// TIA Portal project "KWT_80621" (V14)

(* hardware
DEVICE "S7-1200-Station_1"  S7-1200 Station
   slot 0: "Baugruppenträger_0"  S7-1200 Rack  Rack  V1.0
   slot 1: "PLC_1"  CPU 1214C DC/DC/DC  6ES7 214-1AG40-0XB0  V4.2
   slot 2: "DI 16/DQ 16x24VDC_1"  6ES7 223-1BL32-0XB0  V2.0
   slot 3: "DI 16x24VDC_1"  6ES7 221-1BH32-0XB0  V2.0
   slot 4: "AI 4x13BIT_1"  6ES7 231-4HD32-0XB0  V2.0
   slot 5: "AQ 4x14BIT_1"  6ES7 232-4HD32-0XB0  V2.0
DEVICE "HMI_1"  KTP1200 Basic PN
   slot 0: "KTP1200 Basic PN"  KTP1200 Basic PN  6AV2 123-2MB03-0AX0  14.0.1.0
   slot 1: "HMI_RT_1"  KTP1200 Basic PN  6AV2 123-2MB03-0AX0  14.0.1.0
   slot 5: "HMI_1.IE_CP_1"  PROFINET Interface  14.0.1.0
      slot 1: "PROFINET Schnittstelle_1"  PROFINET Interface
         slot 1: "Port_1"  Port
*)

// ===== PLC "PLC_1"  CPU 1214C DC/DC/DC =====

VAR_GLOBAL   // PLC tag table "Default tag table"
   "System_Byte" AT %MB1 : Byte;
   "FirstScan" AT %M1.0 : Bool;
   "DiagStatusUpdate" AT %M1.1 : Bool;
   "AlwaysTRUE" AT %M1.2 : Bool;
   "AlwaysFALSE" AT %M1.3 : Bool;
   "Clock_Byte" AT %MB0 : Byte;
   "Clock_10Hz" AT %M0.0 : Bool;
   "Clock_5Hz" AT %M0.1 : Bool;
   "Clock_2.5Hz" AT %M0.2 : Bool;
   "Clock_2Hz" AT %M0.3 : Bool;
   "Clock_1.25Hz" AT %M0.4 : Bool;
   "Clock_1Hz" AT %M0.5 : Bool;
   "Clock_0.625Hz" AT %M0.6 : Bool;
   "Clock_0.5Hz" AT %M0.7 : Bool;
END_VAR

VAR_GLOBAL CONSTANT   // PLC tag table "Default tag table"
   "MaxAI10Bit" : Int := 27648;   // AI Max 10 Bit
END_VAR

VAR_GLOBAL   // PLC tag table "1~DI_14_DQ_10"
   "Steuerspannung Ein" AT %I0.0 : Bool;
   "Sicherung Ausgänge OK" AT %I0.1 : Bool;
   "KT 1 Ventilator Störung" AT %I0.2 : Bool;   // Kühlturm 1 Ventilator Störung
   "KT 1 Ventilator Betrieb" AT %I0.3 : Bool;   // Kühlturm 1 Ventilator Betrieb
   "KT 1 Ventilator RS" AT %I0.4 : Bool;   // Kühlturm 1 Ventilator Reparaturschalter ein
   "KT 2 Ventilator Störung" AT %I0.5 : Bool;   // Kühlturm 2 Ventilator Störung
   "KT 2 Ventilator Betrieb" AT %I0.6 : Bool;   // Kühlturm 2 Ventilator Betrieb
   "KT 2 Ventilator RS" AT %I0.7 : Bool;   // Kühlturm 2 Ventilator Reparaturschalter ein
   "Werkspumpe 1 Störung" AT %I1.0 : Bool;
   "Werkspumpe 1 Betrieb" AT %I1.1 : Bool;
   "Werkspumpe 2 Störung" AT %I1.2 : Bool;
   "Werkspumpe 2 Betrieb" AT %I1.3 : Bool;
   "Reserve DI1.4" AT %I1.4 : Bool;
   "Reserve DI1.5" AT %I1.5 : Bool;
   "KT 1 Ventilator" AT %Q0.0 : Bool;   // Kühlturm 1 Ventilator
   "KT 2 Ventilator" AT %Q0.1 : Bool;   // Kühlturm 2 Ventilator
   "Werkspumpe 1" AT %Q0.2 : Bool;
   "Werkspumpe 2" AT %Q0.3 : Bool;
   "Kühlwasserpumpe 1" AT %Q0.4 : Bool;
   "Kühlwasserpumpe 2" AT %Q0.5 : Bool;
   "Rundumleuchte Störung" AT %Q0.6 : Bool;
   "Reserve DQ0.7" AT %Q0.7 : Bool;
   "KT 1 Sprührohr-Klappen öffnen" AT %Q1.0 : Bool;   // Kühlturm 1
   "KT 2 Sprührohr-Klappen öffnen" AT %Q1.1 : Bool;   // Kühlturm 2
END_VAR

VAR_GLOBAL   // PLC tag table "2~DI_16_DQ_16x24VDC"
   "Kühlwasserpumpe 1 MSS OK" AT %I8.0 : Bool;   // Kühlwasserpumpe 1 Motorschutzschalter
   "Kühlwasserpumpe 2 MSS OK" AT %I8.1 : Bool;   // Kühlwasserpumpe 2 Motorschutzschalter
   "Ofenpumpe 1 MSS OK" AT %I8.2 : Bool;   // Ofenpumpe 1 Motorschutzschalter
   "Ofenpumpe 2 MSS OK" AT %I8.3 : Bool;   // Ofenpumpe 2 Motorschutzschalter
   "Kühlwasserpumpe 1 Betrieb" AT %I8.4 : Bool;
   "Kühlwasserpumpe 2 Betrieb" AT %I8.5 : Bool;
   "Ofenpumpe 1 Betrieb" AT %I8.6 : Bool;
   "Ofenpumpe 2 Betrieb" AT %I8.7 : Bool;
   "KT 1 Sprührohr-Klappen geöffnet" AT %I9.0 : Bool;   // Kühlturm 1
   "KT 2 Sprührohr-Klappen geöffnet" AT %I9.1 : Bool;   // Kühlturm 2
   "HA 1 Klappe geöffnet" AT %I9.2 : Bool;   // Hebeanlage 1 Klappe geöffnet
   "HA 1 Klappe geschlossen" AT %I9.3 : Bool;   // Hebeanlage 1 Klappe geschlossen Option
   "HA 2 Klappe geöffnet" AT %I9.4 : Bool;   // Hebeanlage 2 Klappe geöffnet
   "HA 2 Klappe geschlossen" AT %I9.5 : Bool;   // Hebeanlage 2 Klappe geschlossen Option
   "Reserve DI9.6" AT %I9.6 : Bool;
   "Reserve DI9.7" AT %I9.7 : Bool;
   "HA 1 Klappe Freigabe" AT %Q8.0 : Bool;   // Hebeanlage 1 Klappe Freigabe
   "HA 2 Klappe Freigabe" AT %Q8.1 : Bool;   // Hebeanlage 2 Klappe Freigabe
   "Ofenpumpe 1" AT %Q8.2 : Bool;
   "Ofenpumpe 2" AT %Q8.3 : Bool;
   "Reserve DQ8.4" AT %Q8.4 : Bool;
   "Reserve DQ8.5" AT %Q8.5 : Bool;
   "Reserve DQ8.6" AT %Q8.6 : Bool;
   "Reserve DQ8.7" AT %Q8.7 : Bool;
   "WSB Magnetventil" AT %Q9.0 : Bool;   // Wasserstation Behälter Magnetventil Nachfüllung
   "Reserve DQ9.1" AT %Q9.1 : Bool;
   "Reserve DQ9.2" AT %Q9.2 : Bool;
   "Reserve DQ9.3" AT %Q9.3 : Bool;
   "Reserve DQ9.4" AT %Q9.4 : Bool;
   "Reserve DQ9.5" AT %Q9.5 : Bool;
   "Reserve DQ9.6" AT %Q9.6 : Bool;
   "Reserve DQ9.7" AT %Q9.7 : Bool;
END_VAR

VAR_GLOBAL   // PLC tag table "3~DI_16x24VDC"
   "Absalzanlage läuft" AT %I12.0 : Bool;   // Absalzanlage Umwälzpumpe läuft
   "WSB OUT1" AT %I12.1 : Bool;   // Wasserstation Behälter Füllstand binär Bit 0
   "WSB OUT2" AT %I12.2 : Bool;   // Wasserstation Behälter Füllstand binär Bit 1
   "WSB OUT3" AT %I12.3 : Bool;   // Wasserstation Behälter Füllstand binär Bit 2
   "WSB OUT4" AT %I12.4 : Bool;   // Wasserstation Behälter Füllstand binär Bit 3
   "Reserve DI12.5" AT %I12.5 : Bool;
   "Reserve DI12.6" AT %I12.6 : Bool;
   "Reserve DI12.7" AT %I12.7 : Bool;
   "Reserve DI13.0" AT %I13.0 : Bool;
   "Reserve DI13.1" AT %I13.1 : Bool;
   "Reserve DI13.2" AT %I13.2 : Bool;
   "Reserve DI13.3" AT %I13.3 : Bool;
   "Reserve DI13.4" AT %I13.4 : Bool;
   "Reserve DI13.5" AT %I13.5 : Bool;
   "Reserve DI13.6" AT %I13.6 : Bool;
   "Reserve DI13.7" AT %I13.7 : Bool;
   "WSB OUT1 M" AT %M12.0 : Bool;   // Wasserstation Behälter Füllstand binär Bit 0
   "WSB OUT2 M" AT %M12.1 : Bool;   // Wasserstation Behälter Füllstand binär Bit 1
   "WSB OUT3 M" AT %M12.2 : Bool;   // Wasserstation Behälter Füllstand binär Bit 2
   "WSB OUT4 M" AT %M12.3 : Bool;   // Wasserstation Behälter Füllstand binär Bit 3
   "WSB OUT Byte" AT %MB12 : Byte;   // Wasserstation Behälter Füllstand binär Byte
END_VAR

VAR_GLOBAL   // PLC tag table "4~AI_4x13BIT"
   "HA 1 Differenzdruck" AT %IW128 : Int;   // Hebeanlage 1 Differenzdruck Filter
   "HA 2 Differenzdruck" AT %IW130 : Int;   // Hebeanlage 2 Differenzdruck Filter
   "Reserve IW132" AT %IW132 : Int;
   "Reserve IW134" AT %IW134 : Int;
END_VAR

VAR_GLOBAL   // PLC tag table "5~AQ_4"
   "KT 1 Ventilator Sollwert" AT %QW144 : Int;   // Kühlturm 1 Sollwert
   "KT 2 Ventilator Sollwert" AT %QW146 : Int;   // Kühlturm 2 Sollwert
   "HA 1 Klappe Durchflußmenge" AT %QW148 : Int;   // Hebeanlage 1 Klappe Durchflußmenge
   "HA 2 Klappe Durchflußmenge" AT %QW150 : Int;   // Hebeanlage 2 Klappe Durchflußmenge
END_VAR

VAR_GLOBAL   // PLC tag table "1~AI_2"
   "Vorlauftemperatur Werk" AT %IW64 : Int;
   "Vorlauftemperatur Ofen" AT %IW66 : Int;
END_VAR

TYPE "RTM_MODE"
   STRUCT
      FETCH : Byte := 16#0;   // 0: Read out (the status is then written to CQ and the current value to CV). After the operating hours counter has reached (2^31) - 1 hours, it stops at the highest value that can be displayed and outputs an "Overflow" error message.
      START : Byte := 16#1;   // 1: start (at the last counter value)
      STOP : Byte := 16#2;   // 2: stop
      SET : Byte := 16#4;   // 4: set to the value specified in the parameter PV
      SET_START : Byte := 16#5;   // 5: set to the value specified in the parameter PV and start
      SET_STOP : Byte := 16#6;   // 6: set to the value specified in the parameter PV and stop
      SAVE_MC : Byte := 16#7;   // 7: save all RTM values in the CPU to the MC (Memory Card)
   END_STRUCT;
END_TYPE

DATA_BLOCK "Main_DB"   // DB1
{ S7_Optimized_Access := 'TRUE' }
AUTHOR : Searinox(Gerrit_Vogtlaender)
FAMILY : AKK
VERSION : 0.1
// stored: InstanceOfName MainInstane
"MainInstane"
BEGIN
END_DATA_BLOCK

DATA_BLOCK "Retain_DB"   // DB2
{ S7_Optimized_Access := 'TRUE' }
AUTHOR : Searinox
VERSION : 0.1
   VAR RETAIN
      Settings : Struct
         MaxPressureDeltaPerc1 : Int := 50;   // Maximum pressure difference in percent before alarm
         MaxPressureDeltaPerc2 : Int := 50;   // Maximum pressure difference in percent before alarm
         MaxTempTransgression : Real := 4.0;   // Maximum temperature overrun of setpoint in centigrade before alarm
      END_STRUCT;
   END_VAR
BEGIN
END_DATA_BLOCK

FUNCTION_BLOCK "MainInstane"   // FB1, SCL
{ S7_Optimized_Access := 'TRUE' }
AUTHOR : Searinox(Gerrit_Vogtlaender)
FAMILY : AKK
VERSION : 0.1
   VAR
      AlwaysRUN : "AlwaysRUN";
      Auto : "Auto";
      Hand : "Hand";
      AutoMode : Bool := true;
      FlowTemperaturePlant : Real;
      FlowTemperatureFurnace : Real;
   END_VAR
   VAR RETAIN
      HMI : Struct
         StorageTankLevel : Struct
            P1 : Int := 14;   // position 1, e.g. maximum value reached
            P2 : Int := 6;   // position 2, e.g. upper preset value reached
            P3 : Int := 4;   // position 3, e.g. lower preset value reached
            P4 : Int := 2;   // position 4, e.g. minimum value reached
         END_STRUCT;
         StorageTankRefill : Bool;
      END_STRUCT;
   END_VAR
BEGIN
   #AlwaysRUN();

   IF NOT "Steuerspannung Ein" OR NOT "Sicherung Ausgänge OK" THEN
       #AutoMode := 0;
       "KT 1 Ventilator" := 0;
       "KT 2 Ventilator" := 0;
       "Werkspumpe 1" := 0;
       "Werkspumpe 2" := 0;
       "Kühlwasserpumpe 1" := 0;
       "Kühlwasserpumpe 2" := 0;
       //"Rundumleuchte Störung" := 0;
       "Reserve DQ0.7" := 0;
       "KT 1 Sprührohr-Klappen öffnen" := 0;
       "KT 2 Sprührohr-Klappen öffnen" := 0;
       "HA 1 Klappe Freigabe" := 0;
       "HA 2 Klappe Freigabe" := 0;
       "Ofenpumpe 1" := 0;
       "Ofenpumpe 2" := 0;
       "Reserve DQ8.4" := 0;
       "Reserve DQ8.5" := 0;
       "Reserve DQ8.6" := 0;
       "Reserve DQ8.7" := 0;
       "WSB Magnetventil" := 0;
       "Reserve DQ9.1" := 0;
       "Reserve DQ9.2" := 0;
       "Reserve DQ9.3" := 0;
       "Reserve DQ9.4" := 0;
       "Reserve DQ9.5" := 0;
       "Reserve DQ9.6" := 0;
       "Reserve DQ9.7" := 0;
   END_IF;

   IF #AutoMode THEN
       #Auto();
   ELSE
       #Hand();
   END_IF;
END_FUNCTION_BLOCK

FUNCTION_BLOCK "Alarm"   // FB2, SCL
{ S7_Optimized_Access := 'TRUE' }
AUTHOR : Searinox
VERSION : 0.1
   VAR
      "Steuerspannung Ein" : Int;
      "Sicherung Ausgänge OK" : Int;
      "KT 1 Ventilator Störung" : Int;
      "KT 1 Ventilator RS" : Int;
      "KT 2 Ventilator Störung" : Int;
      "KT 2 Ventilator RS" : Int;
      "Werkspumpe 1 Störung" : Int;
      "Werkspumpe 2 Störung" : Int;
      "Kühlwasserpumpe 1 MSS OK" : Int;
      "Kühlwasserpumpe 2 MSS OK" : Int;
      "Ofenpumpe 1 MSS OK" : Int;
      "Ofenpumpe 2 MSS OK" : Int;
      s_alarms : Int;
      FlowTemperaturePlant : Int;
      FlowTemperatureFurnace : Int;
      "HA 1 Differenzdruck" : Int;
      "HA 2 Differenzdruck" : Int;
      SurgeTankRunDry : Int;
      SurgeTankOverflow : Int;
   END_VAR
   VAR_TEMP
      PressureDeltaPerc1 : Int;
      PressureDeltaPerc2 : Int;
   END_VAR
BEGIN
   REGION bool
       #"Steuerspannung Ein" := BOOL_TO_INT(NOT "Steuerspannung Ein");
       #"Sicherung Ausgänge OK" := BOOL_TO_INT(NOT "Sicherung Ausgänge OK");
       #"KT 1 Ventilator Störung" := BOOL_TO_INT("KT 1 Ventilator Störung");
       #"KT 2 Ventilator Störung" := BOOL_TO_INT("KT 2 Ventilator Störung");
       #"KT 1 Ventilator RS" := BOOL_TO_INT(NOT "KT 1 Ventilator RS");
       #"KT 2 Ventilator RS" := BOOL_TO_INT(NOT "KT 2 Ventilator RS");
       #"Werkspumpe 1 Störung" := BOOL_TO_INT("Werkspumpe 1 Störung");
       #"Werkspumpe 2 Störung" := BOOL_TO_INT("Werkspumpe 2 Störung");
       #"Kühlwasserpumpe 1 MSS OK" := BOOL_TO_INT(NOT "Kühlwasserpumpe 1 MSS OK");
       #"Kühlwasserpumpe 2 MSS OK" := BOOL_TO_INT(NOT "Kühlwasserpumpe 2 MSS OK");
       #"Ofenpumpe 1 MSS OK" := BOOL_TO_INT(NOT "Ofenpumpe 1 MSS OK");
       #"Ofenpumpe 2 MSS OK" := BOOL_TO_INT(NOT "Ofenpumpe 2 MSS OK");
   END_REGION
   REGION analog
       // temperatures
       #FlowTemperaturePlant := BOOL_TO_INT("Main_DB".FlowTemperaturePlant >= ("Main_DB".Auto.s_Max + "Retain_DB".Settings.MaxTempTransgression));
       #FlowTemperatureFurnace := BOOL_TO_INT("Main_DB".FlowTemperatureFurnace >= ("Main_DB".Auto.s_Max + "Retain_DB".Settings.MaxTempTransgression));
       // pressures
       #PressureDeltaPerc1 := "ScaleValueInt"(VALUE := "HA 1 Differenzdruck",
                                                XMIN := 0, XMAX := "MaxAI10Bit",
                                                YMIN := 0, YMAX := 100);
       #"HA 1 Differenzdruck" := BOOL_TO_INT(#PressureDeltaPerc1 >= "Retain_DB".Settings.MaxPressureDeltaPerc1);
       #PressureDeltaPerc2 := "ScaleValueInt"(VALUE := "HA 2 Differenzdruck",
                                                XMIN := 0, XMAX := "MaxAI10Bit",
                                                YMIN := 0, YMAX := 100);
       #"HA 2 Differenzdruck" := BOOL_TO_INT(#PressureDeltaPerc2 >= "Retain_DB".Settings.MaxPressureDeltaPerc2);

       #SurgeTankRunDry := BOOL_TO_INT("WSB OUT Byte" <= "Main_DB".HMI.StorageTankLevel.P4);
       #SurgeTankOverflow := BOOL_TO_INT("WSB OUT Byte" >= "Main_DB".HMI.StorageTankLevel.P1);
   END_REGION

   #s_alarms := 0;
   #s_alarms += #"Steuerspannung Ein";
   #s_alarms += #"Sicherung Ausgänge OK";
   #s_alarms += #"KT 1 Ventilator Störung";
   #s_alarms += #"KT 1 Ventilator RS";
   #s_alarms += #"KT 2 Ventilator Störung";
   #s_alarms += #"KT 2 Ventilator RS";
   #s_alarms += #"Werkspumpe 1 Störung";
   #s_alarms += #"Werkspumpe 2 Störung";
   #s_alarms += #"Kühlwasserpumpe 1 MSS OK";
   #s_alarms += #"Kühlwasserpumpe 2 MSS OK";
   #s_alarms += #"Ofenpumpe 1 MSS OK";
   #s_alarms += #"Ofenpumpe 2 MSS OK";
   #s_alarms += #FlowTemperaturePlant;
   #s_alarms += #FlowTemperatureFurnace;
   #s_alarms += #"HA 1 Differenzdruck";
   #s_alarms += #"HA 2 Differenzdruck";
   #s_alarms += #SurgeTankRunDry;
   #s_alarms += #SurgeTankOverflow;

   "Rundumleuchte Störung" := #s_alarms > 0;


   // heizung klappen & endschalter offen zu 
   //Trockenlauf & Überlauf
   //ZU-Klappen 1 geöffnet
END_FUNCTION_BLOCK

FUNCTION_BLOCK "AlwaysRUN"   // FB10, SCL
{ S7_Optimized_Access := 'TRUE' }
AUTHOR : Searinox(Gerrit_Vogtlaender)
FAMILY : AKK
VERSION : 0.1
   VAR
      ScaleAnalogValues : "ScaleAnalogValues";
      RuntimeMeters : "RuntimeMeters";
      Alarm : "Alarm";
      IEC_TMR_0 : IEC_TIMER;
      StorageTankRefill : Bool;
      StorageTankRefillPt : Time := T#5s;
   END_VAR
   VAR_TEMP
      StorageTankRefillEt : Time;
   END_VAR
BEGIN
   #ScaleAnalogValues(i_Vorlauftemp := "Vorlauftemperatur Werk",
                      i_Ruecklauftemp := "Vorlauftemperatur Ofen",
                      o_Vorlauftemp => "Main_DB".FlowTemperaturePlant,
                      o_Ruecklauftemp => "Main_DB".FlowTemperatureFurnace);

   #RuntimeMeters();

   "WSB OUT1 M" := "WSB OUT1";
   "WSB OUT2 M" := "WSB OUT2";
   "WSB OUT3 M" := "WSB OUT3";
   "WSB OUT4 M" := "WSB OUT4";

   #Alarm();

   #IEC_TMR_0.TOF(IN := #StorageTankRefill,
                  PT := #StorageTankRefillPt,
                  Q => "WSB Magnetventil",
                  ET => #StorageTankRefillEt);
END_FUNCTION_BLOCK

FUNCTION_BLOCK "Auto"   // FB20, SCL
{ S7_Optimized_Access := 'TRUE' }
AUTHOR : Searinox(Gerrit_Vogtlaender)
FAMILY : AKK
VERSION : 0.1
   VAR
      s_Min : Real := 0.0;
   END_VAR
   VAR RETAIN
      s_Max : Real := 27.0;
   END_VAR
   VAR
      Werkskreislauf : "Werkskreislauf";
      Kuehlturmkreislauf : "Kuehlturmkreislauf";
      s_MaxCapMin : Real := 0.0;
      s_MaxCapMax : Real := 100.0;
      s_MaxInitVal : Real := 27.0;
      s_MinToMaxZone : Real := 2.0;
      s_strang : Bool;
      Hebeanlage : "Hebeanlage";
   END_VAR
   VAR_TEMP
      t_ret_val : Int;
      t_dtl_out : DTL;
   END_VAR
BEGIN
   #t_ret_val := RD_SYS_T(#t_dtl_out);
   #s_strang := #t_dtl_out.DAY MOD 2 = 0;

   "Main_DB".AlwaysRUN.StorageTankRefill := "WSB OUT Byte" <= "Main_DB".HMI.StorageTankLevel.P2;

   #Werkskreislauf(i_Strang := #s_strang,
                   i_Betrieb1 := "Werkspumpe 1 Betrieb",
                   i_Betrieb2 := "Werkspumpe 2 Betrieb",
                   i_Stoerung1 := "Werkspumpe 1 Störung",
                   i_Stoerung2 := "Werkspumpe 2 Störung",
                   o_Pumpe1 => "Werkspumpe 1",
                   o_Pumpe2 => "Werkspumpe 2");

   #Kuehlturmkreislauf(i_Strang := #s_strang,
                       i_Vorlauftemperatur := "Main_DB".FlowTemperaturePlant,
                       i_Min := #s_Min,
                       i_Max := #s_Max,
                       i_BetriebP1 := "Kühlwasserpumpe 1 Betrieb",
                       i_BetriebP2 := "Kühlwasserpumpe 2 Betrieb",
                       i_StoerungP1 := NOT "Kühlwasserpumpe 1 MSS OK",
                       i_StoerungP2 := NOT "Kühlwasserpumpe 2 MSS OK",
                       i_AbsalzPulse := "Absalzanlage läuft",
                       i_ZuKlappen1offen := "KT 1 Sprührohr-Klappen geöffnet",
                       i_ZuKlappen2offen := "KT 2 Sprührohr-Klappen geöffnet",
                       o_Pumpe3 => "Kühlwasserpumpe 1",
                       o_Pumpe4 => "Kühlwasserpumpe 2",
                       o_Ventilator1 => "KT 1 Ventilator",
                       o_Ventilator2 => "KT 2 Ventilator",
                       o_Ventilator1Sollwert => "KT 1 Ventilator Sollwert",
                       o_Ventilator2Sollwert => "KT 2 Ventilator Sollwert",
                       o_ZuKlappen1oeffnen => "KT 1 Sprührohr-Klappen öffnen",
                       o_ZuKlappen2oeffnen => "KT 2 Sprührohr-Klappen öffnen");

   IF #s_Max < #s_MaxCapMin OR #s_Max > #s_MaxCapMax THEN
       #s_Max := #s_MaxInitVal;
   END_IF;

   #s_Min := #s_Max - #s_MinToMaxZone;

   IF "AlwaysTRUE" THEN
       #Hebeanlage(Strang := #s_strang,
                   Temp := "Main_DB".FlowTemperatureFurnace,
                   TempMin := #s_Min,
                   TempMax := #s_Max + 1,
                   Motorschutzschalter_H1 := NOT "Ofenpumpe 1 MSS OK",
                   Motorschutzschalter_H2 := NOT "Ofenpumpe 2 MSS OK",
                   Betrieb_P1 := "Ofenpumpe 1 Betrieb",
                   Betrieb_P2 := "Ofenpumpe 2 Betrieb",
                   "H1 Klappe geöffnet" := "HA 1 Klappe geöffnet",
                   "H2 Klappe geöffnet" := "HA 2 Klappe geöffnet",
                   "Behälter Trockenlaufschutz" := "WSB OUT1",
                   "Behälter Pumpe ein" := "WSB OUT2",
                   "Behälter Pumpe aus" := "WSB OUT3",
                   "Behälter Überlauf" := "WSB OUT4",
                   "H1 Differenzdruck" := "HA 1 Differenzdruck",
                   "H2 Differenzdruck" := "HA 2 Differenzdruck",
                   "Hebeanlage 1 öffnen" => "HA 1 Klappe Freigabe",
                   "Hebeanlage 2 öffnen" => "HA 2 Klappe Freigabe",
                   Pumpe_H1 => "Ofenpumpe 1",
                   Pumpe_H2 => "Ofenpumpe 2",
                   H1_Durchflußmenge => "HA 1 Klappe Durchflußmenge",
                   H2_Durchflußmenge => "HA 2 Klappe Durchflußmenge");
   END_IF;
END_FUNCTION_BLOCK

FUNCTION_BLOCK "Hand"   // FB30, SCL
{ S7_Optimized_Access := 'TRUE' }
AUTHOR : Searinox(Gerrit_Vogtlaender)
FAMILY : AKK
VERSION : 0.1
   VAR
      static_Vent1SollP : Int;
      static_Vent2SollP : Int;
   END_VAR
BEGIN
   "KT 1 Ventilator Sollwert" := "ScaleValueInt"(VALUE := #static_Vent1SollP, XMIN := 0, XMAX := 100, YMIN := 0, YMAX := "MaxAI10Bit");
   "KT 2 Ventilator Sollwert" := "ScaleValueInt"(VALUE := #static_Vent2SollP, XMIN := 0, XMAX := 100, YMIN := 0, YMAX := "MaxAI10Bit");

   "Main_DB".AlwaysRUN.StorageTankRefill :=
   "Main_DB".HMI.StorageTankRefill AND "WSB OUT Byte" <= "Main_DB".HMI.StorageTankLevel.P2;
END_FUNCTION_BLOCK

FUNCTION_BLOCK "ScaleAnalogValues"   // FB100, SCL
{ S7_Optimized_Access := 'TRUE' }
AUTHOR : Searinox(Gerrit_Vogtlaender)
FAMILY : AKK
VERSION : 0.1
   VAR_INPUT
      i_Vorlauftemp : Int;
      i_Ruecklauftemp : Int;
   END_VAR
   VAR_OUTPUT
      o_Vorlauftemp : Real;
      o_Ruecklauftemp : Real;
   END_VAR
BEGIN
   #o_Vorlauftemp := "Scale_PT100"(#i_Vorlauftemp);
   #o_Ruecklauftemp := "Scale_PT100"(#i_Ruecklauftemp);
END_FUNCTION_BLOCK

FUNCTION_BLOCK "RuntimeMeters"   // FB200, SCL
{ S7_Optimized_Access := 'TRUE' }
AUTHOR : Searinox(Gerrit_Vogtlaender)
FAMILY : AKK
VERSION : 0.1
   VAR
      SRTM : Array[0..9] of "SRTM";
   END_VAR
   VAR_TEMP
      i : Int;
      t_CLK : Bool;
   END_VAR
BEGIN
   FOR #i := 0 TO 9 DO
       CASE #i OF
           0:
               #t_CLK := "AlwaysTRUE";
           1:
               #t_CLK := "Werkspumpe 1 Betrieb";
           2:
               #t_CLK := "Werkspumpe 2 Betrieb";
           3:
               #t_CLK := "Kühlwasserpumpe 1 Betrieb";
           4:
               #t_CLK := "Kühlwasserpumpe 2 Betrieb";
           5:
               #t_CLK := "Ofenpumpe 1 Betrieb";
           6:
               #t_CLK := "Ofenpumpe 2 Betrieb";
           7:
               #t_CLK := "KT 1 Ventilator Betrieb";
           8:
               #t_CLK := "KT 2 Ventilator Betrieb";
           9:
               #t_CLK := "AlwaysFALSE";
           ELSE
               #t_CLK := "AlwaysFALSE";
       END_CASE;
       #SRTM[#i]SRTM(i_CLK := #t_CLK,
                 i_NR := INT_TO_UINT(#i));
   END_FOR;
END_FUNCTION_BLOCK

FUNCTION_BLOCK "Werkskreislauf"   // FB300, SCL
{ S7_Optimized_Access := 'TRUE' }
AUTHOR : Searinox(Gerrit_Vogtlaender)
FAMILY : AKK
VERSION : 0.1
   VAR_INPUT
      i_Strang : Bool;
      i_Betrieb1 : Bool;
      i_Betrieb2 : Bool;
      i_Stoerung1 : Bool;   // Störung
      i_Stoerung2 : Bool;   // Störung
   END_VAR
   VAR_OUTPUT
      o_Pumpe1 : Bool;
      o_Pumpe2 : Bool;
   END_VAR
   VAR
      s_p1 : Bool;
      s_p2 : Bool;
      s_Nachlaufzeit : Time := T#10S;
      Baustein_1 : "Baustein_1";
   END_VAR
BEGIN
   #Baustein_1(i_strang := #i_Strang,
               i_beide := "AlwaysFALSE",
               i_err1 := #i_Stoerung1,
               i_err2 := #i_Stoerung2,
               i_run1 := #i_Betrieb1,
               i_run2 := #i_Betrieb2,
               i_tof_pt := #s_Nachlaufzeit,
               o_p1 => #o_Pumpe1,
               o_p2 => #o_Pumpe2,
               io_s_p1 := #s_p1,
               io_s_p2 := #s_p2);
END_FUNCTION_BLOCK

FUNCTION_BLOCK "Kuehlturmkreislauf"   // FB400, SCL
{ S7_Optimized_Access := 'TRUE' }
AUTHOR : Searinox(Gerrit_Vogtlaender)
FAMILY : AKK
VERSION : 0.1
   VAR_INPUT
      i_Strang : Bool;   // Strang
      i_Vorlauftemperatur : Real;   // Vorlauftemperatur
      i_Min : Real;
      i_Max : Real;
      i_BetriebP1 : Bool;
      i_BetriebP2 : Bool;
      i_StoerungP1 : Bool;
      i_StoerungP2 : Bool;
      i_AbsalzPulse : Bool;
      i_ZuKlappen1offen : Bool;
      i_ZuKlappen2offen : Bool;
   END_VAR
   VAR_OUTPUT
      o_Pumpe3 : Bool;
      o_Pumpe4 : Bool;
      o_Ventilator1 : Bool;
      o_Ventilator2 : Bool;
      o_Ventilator1Sollwert : Int;
      o_Ventilator2Sollwert : Int;
      o_ZuKlappen1oeffnen : Bool;
      o_ZuKlappen2oeffnen : Bool;
   END_VAR
   VAR
      s_Pumpe1 : Bool;
      s_Pumpe2 : Bool;
      s_zu_kalt : Bool;
      s_zu_warm : Bool;
      s_Sollwert : Int;
      s_Ventilator_pt : Time := T#30S;
      s_Beide_Pumpen : Bool;
      s_Nachlaufzeit : Time := T#10S;
      Baustein_1 : "Baustein_1";
      IEC_TMR_0 : IEC_TIMER;
      IEC_TMR_1 : IEC_TIMER;
      s_Ventilator1_ET : Time;
      s_Ventilator2_ET : Time;
      s_SET_POINT_MIN : Int := 0;
      s_SET_POINT_MAX : Int := 27648;
      s_MaxThreshold : Real := 1.0;
      IEC_TMR_2 : IEC_TIMER;
      s_AbsalzPulsePT : Time := T#5m;
      s_AbsalzTP : Bool;
      s_AbsalzPulseET : Time;
   END_VAR
BEGIN
   #s_Beide_Pumpen := #i_Vorlauftemperatur > (#i_Max + #s_MaxThreshold) OR #s_AbsalzTP;

   #Baustein_1(i_strang := #i_Strang,
               i_beide := #s_Beide_Pumpen,
               i_err1 := #i_StoerungP1,
               i_err2 := #i_StoerungP2,
               i_run1 := #i_BetriebP1,
               i_run2 := #i_BetriebP2,
               i_tof_pt := #s_Nachlaufzeit,
               o_p1 => #o_Pumpe3,
               o_p2 => #o_Pumpe4,
               io_s_p1 := #s_Pumpe1,
               io_s_p2 := #s_Pumpe2);

   #IEC_TMR_0.TON(IN := #i_BetriebP1 AND NOT #s_zu_kalt,
                  PT := #s_Ventilator_pt,
                  Q => #o_Ventilator1,
                  ET => #s_Ventilator1_ET);

   #IEC_TMR_1.TON(IN := #i_BetriebP2 AND NOT #s_zu_kalt,
                  PT := #s_Ventilator_pt,
                  Q => #o_Ventilator2,
                  ET => #s_Ventilator2_ET);

   #IEC_TMR_2.TP(IN := #i_AbsalzPulse,
                 PT := #s_AbsalzPulsePT,
                 Q => #s_AbsalzTP,
                 ET => #s_AbsalzPulseET);

   #s_zu_kalt := #i_Vorlauftemperatur <= #i_Min;
   #s_zu_warm := #i_Vorlauftemperatur >= #i_Max;

   IF #s_zu_warm THEN
       #s_Sollwert := #s_SET_POINT_MAX;
   ELSIF #s_zu_kalt THEN
       #s_Sollwert := #s_SET_POINT_MIN;
   ELSE
       #s_Sollwert := "ScaleValueRealToInt"(VALUE := #i_Vorlauftemperatur,
                                            XMIN := #i_Min,
                                            XMAX := #i_Max,
                                            YMIN := #s_SET_POINT_MIN,
                                            YMAX := #s_SET_POINT_MAX);
   END_IF;

   #o_Ventilator1Sollwert := #s_Sollwert;
   #o_Ventilator2Sollwert := #s_Sollwert;
   #o_ZuKlappen1oeffnen := #o_Pumpe3;
   #o_ZuKlappen2oeffnen := #o_Pumpe4;
END_FUNCTION_BLOCK

FUNCTION_BLOCK "Hebeanlage"   // FB500, SCL
{ S7_Optimized_Access := 'TRUE' }
AUTHOR : Searinox(Gerrit_Vogtlaender)
FAMILY : AKK
VERSION : 0.1
   VAR_INPUT
      Strang : Bool;
      Temp : Real;
      TempMin : Real;
      TempMax : Real;
      Motorschutzschalter_H1 : Bool;
      Motorschutzschalter_H2 : Bool;
      Betrieb_P1 : Bool;
      Betrieb_P2 : Bool;
      "H1 Klappe geöffnet" : Bool;
      "H2 Klappe geöffnet" : Bool;
      "Behälter Trockenlaufschutz" : Bool;
      "Behälter Pumpe ein" : Bool;
      "Behälter Pumpe aus" : Bool;
      "Behälter Überlauf" : Bool;
      "H1 Differenzdruck" : Int;
      "H2 Differenzdruck" : Int;
   END_VAR
   VAR_OUTPUT
      "Hebeanlage 1 öffnen" : Bool;
      "Hebeanlage 2 öffnen" : Bool;
      Pumpe_H1 : Bool;
      Pumpe_H2 : Bool;
      H1_Durchflußmenge : Int;
      H2_Durchflußmenge : Int;
   END_VAR
   VAR
      s_P1 : Bool;
      s_P2 : Bool;
      s_Nachlaufzeit : Time := T#10S;
      Baustein_1 : "Baustein_1";
      s_zu_kalt : Bool;
      s_zu_warm : Bool;
      s_Sollwert : Int;
      s_SET_POINT_MIN : Int := 2765;
      s_SET_POINT_MAX : Int := 27648;
      s_Beide_Pumpen : Bool;
      s_MaxThreshold : Real := 1.0;
   END_VAR
BEGIN
   #s_Beide_Pumpen := #Temp > (#TempMax + #s_MaxThreshold);

   #Baustein_1(i_strang := #Strang,
               i_beide := #s_Beide_Pumpen,
               i_err1 := #Motorschutzschalter_H1,
               i_err2 := #Motorschutzschalter_H2,
               i_run1 := #Betrieb_P1,
               i_run2 := #Betrieb_P2,
               i_tof_pt := #s_Nachlaufzeit,
               o_p1 => #Pumpe_H1,
               o_p2 => #Pumpe_H2,
               io_s_p1 := #s_P1,
               io_s_p2 := #s_P2);

   #s_zu_kalt := #Temp <= #TempMin;
   #s_zu_warm := #Temp >= #TempMax;

   IF #s_zu_warm THEN
       #s_Sollwert := #s_SET_POINT_MAX;
   ELSIF #s_zu_kalt THEN
       #s_Sollwert := #s_SET_POINT_MIN;
   ELSE
       #s_Sollwert := "ScaleValueRealToInt"(VALUE := #Temp,
                                            XMIN := #TempMin,
                                            XMAX := #TempMax,
                                            YMIN := #s_SET_POINT_MIN,
                                            YMAX := #s_SET_POINT_MAX);
   END_IF;

   IF #Pumpe_H1 THEN
       #H1_Durchflußmenge := #s_Sollwert;
   ELSE
       #H1_Durchflußmenge := #s_SET_POINT_MIN;
   END_IF;
   IF #Pumpe_H2 THEN
       #H2_Durchflußmenge := #s_Sollwert;
   ELSE
       #H2_Durchflußmenge := #s_SET_POINT_MIN;
   END_IF;

   #"Hebeanlage 1 öffnen" := 1;
   #"Hebeanlage 2 öffnen" := 1;
END_FUNCTION_BLOCK

FUNCTION_BLOCK "Baustein_1"   // FB1000, SCL
{ S7_Optimized_Access := 'TRUE' }
AUTHOR : Searinox(Gerrit_Vogtlaender)
FAMILY : AKK
VERSION : 0.1
   VAR_INPUT
      i_strang : Bool;   // Strang
      i_beide : Bool;   // Beide Pumpen
      i_err1 : Bool;
      i_err2 : Bool;
      i_run1 : Bool;
      i_run2 : Bool;
      i_tof_pt : Time;   // Nachlaufzeit
   END_VAR
   VAR_OUTPUT
      o_p1 : Bool;   // Ausgang P1
      o_p2 : Bool;   // Ausgang P2
   END_VAR
   VAR_IN_OUT
      io_s_p1 : Bool;   // static im caller
      io_s_p2 : Bool;   // static im caller
   END_VAR
   VAR
      i_IEC_TMR_1 : IEC_TIMER;
      i_IEC_TMR_2 : IEC_TIMER;
   END_VAR
   VAR_TEMP
      t_err_p1 : Bool;
      t_err_p2 : Bool;
   END_VAR
BEGIN
   #t_err_p1 := #io_s_p1 AND (#i_err1 OR NOT #i_run1);
   #t_err_p2 := #io_s_p2 AND (#i_err2 OR NOT #i_run2);

   #io_s_p1 := #i_strang = 1 OR #t_err_p2 OR #i_beide;
   #io_s_p2 := #i_strang = 0 OR #t_err_p1 OR #i_beide;

   #i_IEC_TMR_1.TOF(IN := #io_s_p1,
                    PT := #i_tof_pt,
                    Q => #o_p1);
   #i_IEC_TMR_2.TOF(IN := #io_s_p2,
                    PT := #i_tof_pt,
                    Q => #o_p2);
END_FUNCTION_BLOCK

FUNCTION_BLOCK "SRTM"   // FB2000, SCL
TITLE = Simple runtime meter wrapper
{ S7_Optimized_Access := 'TRUE' }
AUTHOR : Searinox(Gerrit_Vogtlaender)
FAMILY : AKK
VERSION : 0.1
   VAR_INPUT
      i_CLK : Bool;   // Incoming signal, the edge of which is to be queried
      i_NR : UInt;   // Number of the operating hours counter
   END_VAR
   VAR
      R_TRIG : R_TRIG;   // Detect positive signal edge
      F_TRIG : F_TRIG;   // Detect negative signal edge
      RTM_MODE : "RTM_MODE";   // Job IDs
      s_MODE : Byte;   // Job ID
      s_PV : DInt;   // New value for the operating hours counter
      s_CQ : Bool;   // Status of the operating hours counter (1: running)
      s_RET_VAL : Int;   // If an error occurs while the instruction is being executed, the return value contains an error code.
      s_CV : DInt;   // Current value of the operating hours counter
   END_VAR
   VAR_TEMP
      t_R_TRIG_Q : Bool;   // Result of positive edge evaluation
      t_F_TRIG_Q : Bool;   // Result of negative edge evaluation
   END_VAR
BEGIN
   #R_TRIG(CLK := #i_CLK,
           Q => #t_R_TRIG_Q);
   #F_TRIG(CLK := #i_CLK,
           Q => #t_F_TRIG_Q);

   IF #t_R_TRIG_Q THEN
       #s_MODE := #RTM_MODE.START;
   ELSIF #t_F_TRIG_Q THEN
       #s_MODE := #RTM_MODE.STOP;
   ELSE
       #s_MODE := #RTM_MODE.FETCH;
   END_IF;

   #s_RET_VAL := RTM(NR := #i_NR,
                     MODE := #s_MODE,
                     PV := #s_PV,
                     CQ => #s_CQ,
                     CV => #s_CV);
END_FUNCTION_BLOCK

FUNCTION "Scale_PT100" : Real   // FC1, SCL
{ S7_Optimized_Access := 'TRUE' }
AUTHOR : Searinox(Gerrit_Vogtlaender)
FAMILY : AKK
VERSION : 0.1
   VAR_INPUT
      value : Int;
   END_VAR
   VAR_TEMP
      t_norm : Real;
   END_VAR
BEGIN
   #t_norm := NORM_X(MIN := 0, VALUE := #value, MAX := "MaxAI10Bit");
   #Scale_PT100 := LREAL_TO_REAL(SCALE_X(MIN := 0.0, VALUE := #t_norm, MAX := 100.0));
END_FUNCTION

FUNCTION "ScaleValueInt" : Int   // FC2, SCL
TITLE = ScaleValue
{ S7_Optimized_Access := 'TRUE' }
AUTHOR : Searinox(Gerrit_Vogtlaender)
FAMILY : AKK
NAME : 1337
VERSION : 0.1
// Der Baustein liefert einen linearen Zusammenhang zwischen dem Wert am Eingang I1 und dem Wert am Ausgang QV. Der Ausgangswert wird durch die beiden Koordinatenpaare X1, Y1 und X2, Y2 definiert.
   VAR_INPUT
      VALUE : Int;   // Eingangswert
      XMIN : Int;   // Stützpunkt 1
      XMAX : Int;   // Stützpunkt 2
      YMIN : Int;   // Stützpunkt 1
      YMAX : Int;   // Stützpunkt 2
   END_VAR
   VAR_TEMP
      t_norm : Real;
   END_VAR
   // Ret_Val : beinhaltet den skalierten Eingangswert
BEGIN
   #t_norm := NORM_X(MIN := #XMIN, VALUE := #VALUE, MAX := #XMAX);
   #ScaleValueInt := SCALE_X(MIN := #YMIN, VALUE := #t_norm, MAX := #YMAX);
END_FUNCTION

FUNCTION "ScaleValueRealToInt" : Int   // FC3, SCL
TITLE = ScaleValue
{ S7_Optimized_Access := 'TRUE' }
AUTHOR : Searinox(Gerrit_Vogtlaender)
FAMILY : AKK
NAME : 1337
VERSION : 0.1
// Der Baustein liefert einen linearen Zusammenhang zwischen dem Wert am Eingang I1 und dem Wert am Ausgang QV. Der Ausgangswert wird durch die beiden Koordinatenpaare X1, Y1 und X2, Y2 definiert.
   VAR_INPUT
      VALUE : Real;   // Eingangswert
      XMIN : Real;   // Stützpunkt 1
      XMAX : Real;   // Stützpunkt 2
      YMIN : Int;   // Stützpunkt 1
      YMAX : Int;   // Stützpunkt 2
   END_VAR
   VAR_TEMP
      t_norm : Real;
   END_VAR
BEGIN
   #t_norm := NORM_X(MIN := #XMIN, VALUE := #VALUE, MAX := #XMAX);
   #ScaleValueRealToInt := SCALE_X(MIN := #YMIN, VALUE := #t_norm, MAX := #YMAX);
END_FUNCTION

ORGANIZATION_BLOCK "Main"   // OB1, SCL, ProgramCycle
TITLE = "Main Program Sweep (Cycle)"
{ S7_Optimized_Access := 'TRUE' }
AUTHOR : Searinox(Gerrit_Vogtlaender)
FAMILY : AKK
VERSION : 0.1
BEGIN
   "Main_DB"();
END_ORGANIZATION_BLOCK

(* ===== HMI "HMI_RT_1" =====
system functions are stored by id; their names below are inferred from use
connection "HMI_Verbindung_1": ETHERNET, SMART_S7_1200_OMS

HMI tags "Default tag table"
   "Variable_Bildnummer" : UInt, internal
   "Main_DB_FlowTemperaturePlant" : Real = PLC Main_DB.FlowTemperaturePlant, 1 s
   "Main_DB_FlowTemperatureFurnace" : Real = PLC Main_DB.FlowTemperatureFurnace, 1 s
   "Main_DB_AutoMode" : Bool = PLC Main_DB.AutoMode, 1 s
   "Main_DB_Hand_static_Vent1SollP" : Int = PLC Main_DB.Hand.static_Vent1SollP, 1 s
   "Main_DB_Hand_static_Vent2SollP" : Int = PLC Main_DB.Hand.static_Vent2SollP, 1 s
   "Main_DB_Auto_s_Max" : Real = PLC Main_DB.Auto.s_Max, 1 s
   "WSB OUT Byte" : Byte = PLC "WSB OUT Byte" AT %MB12, 1 s
   "Main_DB_HMI_StorageTankLevel_P1" : Int = PLC Main_DB.HMI.StorageTankLevel.P1, 1 s
   "Main_DB_HMI_StorageTankLevel_P2" : Int = PLC Main_DB.HMI.StorageTankLevel.P2, 1 s
   "Main_DB_HMI_StorageTankLevel_P3" : Int = PLC Main_DB.HMI.StorageTankLevel.P3, 1 s
   "Main_DB_HMI_StorageTankLevel_P4" : Int = PLC Main_DB.HMI.StorageTankLevel.P4, 1 s
   "Main_DB_HMI_StorageTankRefill" : Bool = PLC Main_DB.HMI.StorageTankRefill, 1 s
   "Main_DB_AlwaysRUN_Alarm_Sicherung Ausgänge OK" : Int = PLC Main_DB.AlwaysRUN.Alarm."Sicherung Ausgänge OK", 1 s
   "Main_DB_AlwaysRUN_Alarm_KT 1 Ventilator Störung" : Int = PLC Main_DB.AlwaysRUN.Alarm."KT 1 Ventilator Störung", 1 s
   "Main_DB_AlwaysRUN_Alarm_KT 1 Ventilator RS" : Int = PLC Main_DB.AlwaysRUN.Alarm."KT 1 Ventilator RS", 1 s
   "Main_DB_AlwaysRUN_Alarm_KT 2 Ventilator Störung" : Int = PLC Main_DB.AlwaysRUN.Alarm."KT 2 Ventilator Störung", 1 s
   "Main_DB_AlwaysRUN_Alarm_KT 2 Ventilator RS" : Int = PLC Main_DB.AlwaysRUN.Alarm."KT 2 Ventilator RS", 1 s
   "Main_DB_AlwaysRUN_Alarm_Werkspumpe 1 Störung" : Int = PLC Main_DB.AlwaysRUN.Alarm."Werkspumpe 1 Störung", 1 s
   "Main_DB_AlwaysRUN_Alarm_Werkspumpe 2 Störung" : Int = PLC Main_DB.AlwaysRUN.Alarm."Werkspumpe 2 Störung", 1 s
   "Main_DB_AlwaysRUN_Alarm_Kühlwasserpumpe 1 MSS OK" : Int = PLC Main_DB.AlwaysRUN.Alarm."Kühlwasserpumpe 1 MSS OK", 1 s
   "Main_DB_AlwaysRUN_Alarm_Kühlwasserpumpe 2 MSS OK" : Int = PLC Main_DB.AlwaysRUN.Alarm."Kühlwasserpumpe 2 MSS OK", 1 s
   "Main_DB_AlwaysRUN_Alarm_Ofenpumpe 1 MSS OK" : Int = PLC Main_DB.AlwaysRUN.Alarm."Ofenpumpe 1 MSS OK", 1 s
   "Main_DB_AlwaysRUN_Alarm_Ofenpumpe 2 MSS OK" : Int = PLC Main_DB.AlwaysRUN.Alarm."Ofenpumpe 2 MSS OK", 1 s
   "Main_DB_AlwaysRUN_Alarm_FlowTemperaturePlant" : Int = PLC Main_DB.AlwaysRUN.Alarm.FlowTemperaturePlant, 1 s
   "Main_DB_AlwaysRUN_Alarm_FlowTemperatureFurnace" : Int = PLC Main_DB.AlwaysRUN.Alarm.FlowTemperatureFurnace, 1 s
   "Main_DB_AlwaysRUN_Alarm_HA 1 Differenzdruck" : Int = PLC Main_DB.AlwaysRUN.Alarm."HA 1 Differenzdruck", 1 s
   "Main_DB_AlwaysRUN_Alarm_HA 2 Differenzdruck" : Int = PLC Main_DB.AlwaysRUN.Alarm."HA 2 Differenzdruck", 1 s
   "Main_DB_AlwaysRUN_Alarm_SurgeTankRunDry" : Int = PLC Main_DB.AlwaysRUN.Alarm.SurgeTankRunDry, 1 s
   "Main_DB_AlwaysRUN_Alarm_SurgeTankOverflow" : Int = PLC Main_DB.AlwaysRUN.Alarm.SurgeTankOverflow, 1 s

HMI tags "RuntimeMeters"
   "Main_DB_AlwaysRUN_RuntimeMeters_SRTM{0}_i_CLK" : Bool = PLC Main_DB.AlwaysRUN.RuntimeMeters.SRTM[0].i_CLK, 1 s
   "Main_DB_AlwaysRUN_RuntimeMeters_SRTM{0}_s_CQ" : Bool = PLC Main_DB.AlwaysRUN.RuntimeMeters.SRTM[0].s_CQ, 1 s
   "Main_DB_AlwaysRUN_RuntimeMeters_SRTM{0}_s_CV" : DInt = PLC Main_DB.AlwaysRUN.RuntimeMeters.SRTM[0].s_CV, 1 s
   "Main_DB_AlwaysRUN_RuntimeMeters_SRTM{1}_i_CLK" : Bool = PLC Main_DB.AlwaysRUN.RuntimeMeters.SRTM[1].i_CLK, 1 s
   "Main_DB_AlwaysRUN_RuntimeMeters_SRTM{1}_s_CQ" : Bool = PLC Main_DB.AlwaysRUN.RuntimeMeters.SRTM[1].s_CQ, 1 s
   "Main_DB_AlwaysRUN_RuntimeMeters_SRTM{1}_s_CV" : DInt = PLC Main_DB.AlwaysRUN.RuntimeMeters.SRTM[1].s_CV, 1 s
   "Main_DB_AlwaysRUN_RuntimeMeters_SRTM{2}_i_CLK" : Bool = PLC Main_DB.AlwaysRUN.RuntimeMeters.SRTM[2].i_CLK, 1 s
   "Main_DB_AlwaysRUN_RuntimeMeters_SRTM{2}_s_CQ" : Bool = PLC Main_DB.AlwaysRUN.RuntimeMeters.SRTM[2].s_CQ, 1 s
   "Main_DB_AlwaysRUN_RuntimeMeters_SRTM{2}_s_CV" : DInt = PLC Main_DB.AlwaysRUN.RuntimeMeters.SRTM[2].s_CV, 1 s
   "Main_DB_AlwaysRUN_RuntimeMeters_SRTM{3}_i_CLK" : Bool = PLC Main_DB.AlwaysRUN.RuntimeMeters.SRTM[3].i_CLK, 1 s
   "Main_DB_AlwaysRUN_RuntimeMeters_SRTM{3}_s_CQ" : Bool = PLC Main_DB.AlwaysRUN.RuntimeMeters.SRTM[3].s_CQ, 1 s
   "Main_DB_AlwaysRUN_RuntimeMeters_SRTM{3}_s_CV" : DInt = PLC Main_DB.AlwaysRUN.RuntimeMeters.SRTM[3].s_CV, 1 s
   "Main_DB_AlwaysRUN_RuntimeMeters_SRTM{4}_i_CLK" : Bool = PLC Main_DB.AlwaysRUN.RuntimeMeters.SRTM[4].i_CLK, 1 s
   "Main_DB_AlwaysRUN_RuntimeMeters_SRTM{4}_s_CQ" : Bool = PLC Main_DB.AlwaysRUN.RuntimeMeters.SRTM[4].s_CQ, 1 s
   "Main_DB_AlwaysRUN_RuntimeMeters_SRTM{4}_s_CV" : DInt = PLC Main_DB.AlwaysRUN.RuntimeMeters.SRTM[4].s_CV, 1 s
   "Main_DB_AlwaysRUN_RuntimeMeters_SRTM{5}_i_CLK" : Bool = PLC Main_DB.AlwaysRUN.RuntimeMeters.SRTM[5].i_CLK, 1 s
   "Main_DB_AlwaysRUN_RuntimeMeters_SRTM{5}_s_CQ" : Bool = PLC Main_DB.AlwaysRUN.RuntimeMeters.SRTM[5].s_CQ, 1 s
   "Main_DB_AlwaysRUN_RuntimeMeters_SRTM{5}_s_CV" : DInt = PLC Main_DB.AlwaysRUN.RuntimeMeters.SRTM[5].s_CV, 1 s
   "Main_DB_AlwaysRUN_RuntimeMeters_SRTM{6}_i_CLK" : Bool = PLC Main_DB.AlwaysRUN.RuntimeMeters.SRTM[6].i_CLK, 1 s
   "Main_DB_AlwaysRUN_RuntimeMeters_SRTM{6}_s_CQ" : Bool = PLC Main_DB.AlwaysRUN.RuntimeMeters.SRTM[6].s_CQ, 1 s
   "Main_DB_AlwaysRUN_RuntimeMeters_SRTM{6}_s_CV" : DInt = PLC Main_DB.AlwaysRUN.RuntimeMeters.SRTM[6].s_CV, 1 s
   "Main_DB_AlwaysRUN_RuntimeMeters_SRTM{7}_i_CLK" : Bool = PLC Main_DB.AlwaysRUN.RuntimeMeters.SRTM[7].i_CLK, 1 s
   "Main_DB_AlwaysRUN_RuntimeMeters_SRTM{7}_s_CQ" : Bool = PLC Main_DB.AlwaysRUN.RuntimeMeters.SRTM[7].s_CQ, 1 s
   "Main_DB_AlwaysRUN_RuntimeMeters_SRTM{7}_s_CV" : DInt = PLC Main_DB.AlwaysRUN.RuntimeMeters.SRTM[7].s_CV, 1 s
   "Main_DB_AlwaysRUN_RuntimeMeters_SRTM{8}_i_CLK" : Bool = PLC Main_DB.AlwaysRUN.RuntimeMeters.SRTM[8].i_CLK, 1 s
   "Main_DB_AlwaysRUN_RuntimeMeters_SRTM{8}_s_CQ" : Bool = PLC Main_DB.AlwaysRUN.RuntimeMeters.SRTM[8].s_CQ, 1 s
   "Main_DB_AlwaysRUN_RuntimeMeters_SRTM{8}_s_CV" : DInt = PLC Main_DB.AlwaysRUN.RuntimeMeters.SRTM[8].s_CV, 1 s
   "Main_DB_AlwaysRUN_RuntimeMeters_SRTM{9}_i_CLK" : Bool = PLC Main_DB.AlwaysRUN.RuntimeMeters.SRTM[9].i_CLK, 1 s
   "Main_DB_AlwaysRUN_RuntimeMeters_SRTM{9}_s_CQ" : Bool = PLC Main_DB.AlwaysRUN.RuntimeMeters.SRTM[9].s_CQ, 1 s
   "Main_DB_AlwaysRUN_RuntimeMeters_SRTM{9}_s_CV" : DInt = PLC Main_DB.AlwaysRUN.RuntimeMeters.SRTM[9].s_CV, 1 s

HMI tags "Scaled"
   "HA 1 Differenzdruck(1)" : Int = PLC "HA 1 Differenzdruck" AT %IW128, 1 s
   "HA 1 Klappe Durchflußmenge(1)" : Int = PLC "HA 1 Klappe Durchflußmenge" AT %QW148, 1 s
   "HA 2 Differenzdruck(1)" : Int = PLC "HA 2 Differenzdruck" AT %IW130, 1 s
   "HA 2 Klappe Durchflußmenge(1)" : Int = PLC "HA 2 Klappe Durchflußmenge" AT %QW150, 1 s
   "Reserve IW132(1)" : Int = PLC "Reserve IW132" AT %IW132, 1 s
   "Reserve IW134(1)" : Int = PLC "Reserve IW134" AT %IW134, 1 s
   "Vorlauftemperatur Ofen(1)" : Int = PLC "Vorlauftemperatur Ofen" AT %IW66, 1 s
   "KT 1 Ventilator Sollwert(1)" : Int = PLC "KT 1 Ventilator Sollwert" AT %QW144, 1 s
   "KT 2 Ventilator Sollwert(1)" : Int = PLC "KT 2 Ventilator Sollwert" AT %QW146, 1 s
   "Vorlauftemperatur Werk(1)" : Int = PLC "Vorlauftemperatur Werk" AT %IW64, 1 s

HMI tags "Q"
   "KT 1 Ventilator" : Bool = PLC "KT 1 Ventilator" AT %Q0.0, 1 s
   "KT 2 Ventilator" : Bool = PLC "KT 2 Ventilator" AT %Q0.1, 1 s
   "Werkspumpe 1" : Bool = PLC "Werkspumpe 1" AT %Q0.2, 1 s
   "Werkspumpe 2" : Bool = PLC "Werkspumpe 2" AT %Q0.3, 1 s
   "Kühlwasserpumpe 1" : Bool = PLC "Kühlwasserpumpe 1" AT %Q0.4, 1 s
   "Kühlwasserpumpe 2" : Bool = PLC "Kühlwasserpumpe 2" AT %Q0.5, 1 s
   "Rundumleuchte Störung" : Bool = PLC "Rundumleuchte Störung" AT %Q0.6, 1 s
   "Reserve DQ0.7" : Bool = PLC "Reserve DQ0.7" AT %Q0.7, 1 s
   "KT 1 Sprührohr-Klappen öffnen" : Bool = PLC "KT 1 Sprührohr-Klappen öffnen" AT %Q1.0, 1 s
   "KT 2 Sprührohr-Klappen öffnen" : Bool = PLC "KT 2 Sprührohr-Klappen öffnen" AT %Q1.1, 1 s
   "HA 1 Klappe Freigabe" : Bool = PLC "HA 1 Klappe Freigabe" AT %Q8.0, 1 s
   "HA 2 Klappe Freigabe" : Bool = PLC "HA 2 Klappe Freigabe" AT %Q8.1, 1 s
   "Ofenpumpe 1" : Bool = PLC "Ofenpumpe 1" AT %Q8.2, 1 s
   "Ofenpumpe 2" : Bool = PLC "Ofenpumpe 2" AT %Q8.3, 1 s
   "Reserve DQ8.4" : Bool = PLC "Reserve DQ8.4" AT %Q8.4, 1 s
   "Reserve DQ8.5" : Bool = PLC "Reserve DQ8.5" AT %Q8.5, 1 s
   "Reserve DQ8.6" : Bool = PLC "Reserve DQ8.6" AT %Q8.6, 1 s
   "Reserve DQ8.7" : Bool = PLC "Reserve DQ8.7" AT %Q8.7, 1 s
   "WSB Magnetventil" : Bool = PLC "WSB Magnetventil" AT %Q9.0, 1 s
   "Reserve DQ9.1" : Bool = PLC "Reserve DQ9.1" AT %Q9.1, 1 s
   "Reserve DQ9.2" : Bool = PLC "Reserve DQ9.2" AT %Q9.2, 1 s
   "Reserve DQ9.3" : Bool = PLC "Reserve DQ9.3" AT %Q9.3, 1 s
   "Reserve DQ9.4" : Bool = PLC "Reserve DQ9.4" AT %Q9.4, 1 s
   "Reserve DQ9.5" : Bool = PLC "Reserve DQ9.5" AT %Q9.5, 1 s
   "Reserve DQ9.6" : Bool = PLC "Reserve DQ9.6" AT %Q9.6, 1 s
   "Reserve DQ9.7" : Bool = PLC "Reserve DQ9.7" AT %Q9.7, 1 s

HMI tags "I"
   "Steuerspannung Ein" : Bool = PLC "Steuerspannung Ein" AT %I0.0, 1 s
   "Sicherung Ausgänge OK" : Bool = PLC "Sicherung Ausgänge OK" AT %I0.1, 1 s
   "KT 1 Ventilator Störung" : Bool = PLC "KT 1 Ventilator Störung" AT %I0.2, 1 s
   "KT 1 Ventilator Betrieb" : Bool = PLC "KT 1 Ventilator Betrieb" AT %I0.3, 1 s
   "KT 1 Ventilator RS" : Bool = PLC "KT 1 Ventilator RS" AT %I0.4, 1 s
   "KT 2 Ventilator Störung" : Bool = PLC "KT 2 Ventilator Störung" AT %I0.5, 1 s
   "KT 2 Ventilator Betrieb" : Bool = PLC "KT 2 Ventilator Betrieb" AT %I0.6, 1 s
   "KT 2 Ventilator RS" : Bool = PLC "KT 2 Ventilator RS" AT %I0.7, 1 s
   "Werkspumpe 1 Störung" : Bool = PLC "Werkspumpe 1 Störung" AT %I1.0, 1 s
   "Werkspumpe 2 Störung" : Bool = PLC "Werkspumpe 2 Störung" AT %I1.2, 1 s
   "Werkspumpe 1 Betrieb" : Bool = PLC "Werkspumpe 1 Betrieb" AT %I1.1, 1 s
   "Werkspumpe 2 Betrieb" : Bool = PLC "Werkspumpe 2 Betrieb" AT %I1.3, 1 s
   "Reserve DI1.5" : Bool = PLC "Reserve DI1.5" AT %I1.5, 1 s
   "Kühlwasserpumpe 2 MSS OK" : Bool = PLC "Kühlwasserpumpe 2 MSS OK" AT %I8.1, 1 s
   "Ofenpumpe 1 MSS OK" : Bool = PLC "Ofenpumpe 1 MSS OK" AT %I8.2, 1 s
   "Ofenpumpe 2 MSS OK" : Bool = PLC "Ofenpumpe 2 MSS OK" AT %I8.3, 1 s
   "Reserve DI1.4" : Bool = PLC "Reserve DI1.4" AT %I1.4, 1 s
   "Kühlwasserpumpe 1 MSS OK" : Bool = PLC "Kühlwasserpumpe 1 MSS OK" AT %I8.0, 1 s
   "Kühlwasserpumpe 1 Betrieb" : Bool = PLC "Kühlwasserpumpe 1 Betrieb" AT %I8.4, 1 s
   "Reserve DI12.6" : Bool = PLC "Reserve DI12.6" AT %I12.6, 1 s
   "Reserve DI12.7" : Bool = PLC "Reserve DI12.7" AT %I12.7, 1 s
   "Reserve DI13.0" : Bool = PLC "Reserve DI13.0" AT %I13.0, 1 s
   "Reserve DI13.1" : Bool = PLC "Reserve DI13.1" AT %I13.1, 1 s
   "Reserve DI13.2" : Bool = PLC "Reserve DI13.2" AT %I13.2, 1 s
   "Reserve DI13.3" : Bool = PLC "Reserve DI13.3" AT %I13.3, 1 s
   "Reserve DI13.4" : Bool = PLC "Reserve DI13.4" AT %I13.4, 1 s
   "Reserve DI13.5" : Bool = PLC "Reserve DI13.5" AT %I13.5, 1 s
   "Reserve DI13.6" : Bool = PLC "Reserve DI13.6" AT %I13.6, 1 s
   "Reserve DI13.7" : Bool = PLC "Reserve DI13.7" AT %I13.7, 1 s
   "Kühlwasserpumpe 2 Betrieb" : Bool = PLC "Kühlwasserpumpe 2 Betrieb" AT %I8.5, 1 s
   "Ofenpumpe 1 Betrieb" : Bool = PLC "Ofenpumpe 1 Betrieb" AT %I8.6, 1 s
   "Ofenpumpe 2 Betrieb" : Bool = PLC "Ofenpumpe 2 Betrieb" AT %I8.7, 1 s
   "WSB OUT1" : Bool = PLC "WSB OUT1" AT %I12.1, 1 s
   "WSB OUT2" : Bool = PLC "WSB OUT2" AT %I12.2, 1 s
   "WSB OUT3" : Bool = PLC "WSB OUT3" AT %I12.3, 1 s
   "WSB OUT4" : Bool = PLC "WSB OUT4" AT %I12.4, 1 s
   "Reserve DI12.5" : Bool = PLC "Reserve DI12.5" AT %I12.5, 1 s
   "KT 1 Sprührohr-Klappen geöffnet" : Bool = PLC "KT 1 Sprührohr-Klappen geöffnet" AT %I9.0, 1 s
   "KT 2 Sprührohr-Klappen geöffnet" : Bool = PLC "KT 2 Sprührohr-Klappen geöffnet" AT %I9.1, 1 s
   "HA 1 Klappe geöffnet" : Bool = PLC "HA 1 Klappe geöffnet" AT %I9.2, 1 s
   "HA 1 Klappe geschlossen" : Bool = PLC "HA 1 Klappe geschlossen" AT %I9.3, 1 s
   "Reserve DI9.6" : Bool = PLC "Reserve DI9.6" AT %I9.6, 1 s
   "HA 2 Klappe geschlossen" : Bool = PLC "HA 2 Klappe geschlossen" AT %I9.5, 1 s
   "HA 2 Klappe geöffnet" : Bool = PLC "HA 2 Klappe geöffnet" AT %I9.4, 1 s
   "Reserve DI9.7" : Bool = PLC "Reserve DI9.7" AT %I9.7, 1 s
   "Absalzanlage läuft" : Bool = PLC "Absalzanlage läuft" AT %I12.0, 1 s

HMI tags "IW"
   "Vorlauftemperatur Werk" : Int = PLC "Vorlauftemperatur Werk" AT %IW64, 1 s
   "Vorlauftemperatur Ofen" : Int = PLC "Vorlauftemperatur Ofen" AT %IW66, 1 s
   "HA 1 Differenzdruck" : Int = PLC "HA 1 Differenzdruck" AT %IW128, 1 s
   "HA 2 Differenzdruck" : Int = PLC "HA 2 Differenzdruck" AT %IW130, 1 s
   "Reserve IW132" : Int = PLC "Reserve IW132" AT %IW132, 1 s
   "Reserve IW134" : Int = PLC "Reserve IW134" AT %IW134, 1 s

HMI tags "QW"
   "KT 1 Ventilator Sollwert" : Int = PLC "KT 1 Ventilator Sollwert" AT %QW144, 1 s
   "KT 2 Ventilator Sollwert" : Int = PLC "KT 2 Ventilator Sollwert" AT %QW146, 1 s
   "HA 1 Klappe Durchflußmenge" : Int = PLC "HA 1 Klappe Durchflußmenge" AT %QW148, 1 s
   "HA 2 Klappe Durchflußmenge" : Int = PLC "HA 2 Klappe Durchflußmenge" AT %QW150, 1 s

HMI tags "Alarm"
   "Main_DB_AlwaysRUN_Alarm_Steuerspannung Ein" : Int = PLC Main_DB.AlwaysRUN.Alarm."Steuerspannung Ein", 1 s

discrete alarms
   1: 'NOT AUS', class Errors, trigger "Main_DB_AlwaysRUN_Alarm_Steuerspannung Ein" bit 0
   2: 'Sicherung Ausgänge', class Errors, trigger "Main_DB_AlwaysRUN_Alarm_Sicherung Ausgänge OK" bit 0
   3: 'Kühlturm 1 Ventilator Störung', class Errors, trigger "Main_DB_AlwaysRUN_Alarm_KT 1 Ventilator Störung" bit 0
   4: 'Kühlturm 1 Ventilator Reparaturschalter aus', class Errors, trigger "Main_DB_AlwaysRUN_Alarm_KT 1 Ventilator RS" bit 0
   5: 'Kühlturm 2 Ventilator Störung', class Errors, trigger "Main_DB_AlwaysRUN_Alarm_KT 2 Ventilator Störung" bit 0
   6: 'Kühlturm 2 Ventilator Reparaturschalter aus', class Errors, trigger "Main_DB_AlwaysRUN_Alarm_KT 2 Ventilator RS" bit 0
   7: 'Werkspumpe 1 Störung', class Errors, trigger "Main_DB_AlwaysRUN_Alarm_Werkspumpe 1 Störung" bit 0
   8: 'Werkspumpe 2 Störung', class Errors, trigger "Main_DB_AlwaysRUN_Alarm_Werkspumpe 2 Störung" bit 0
   9: 'Kühlwasserpumpe 1 Motorschutzschalter', class Errors, trigger "Main_DB_AlwaysRUN_Alarm_Kühlwasserpumpe 1 MSS OK" bit 0
   10: 'Kühlwasserpumpe 2 Motorschutzschalter', class Errors, trigger "Main_DB_AlwaysRUN_Alarm_Kühlwasserpumpe 2 MSS OK" bit 0
   11: 'Ofenpumpe 1 Motorschutzschalter', class Errors, trigger "Main_DB_AlwaysRUN_Alarm_Ofenpumpe 1 MSS OK" bit 0
   12: 'Ofenpumpe 2 Motorschutzschalter', class Errors, trigger "Main_DB_AlwaysRUN_Alarm_Ofenpumpe 2 MSS OK" bit 0
   13: 'Vorlauftemperatur Werk zu hoch', class Errors, trigger "Main_DB_AlwaysRUN_Alarm_FlowTemperaturePlant" bit 0
   14: 'Vorlauftemperatur Ofenkühlung zu hoch', class Errors, trigger "Main_DB_AlwaysRUN_Alarm_FlowTemperatureFurnace" bit 0
   15: 'Hebeanlage Filter 1 Differenzdruck zu hoch', class Errors, trigger "Main_DB_AlwaysRUN_Alarm_HA 1 Differenzdruck" bit 0
   16: 'Hebeanlage Filter 2 Differenzdruck zu hoch', class Errors, trigger "Main_DB_AlwaysRUN_Alarm_HA 2 Differenzdruck" bit 0
   17: 'Wasserstation Ausgleichsbehälter läuft trocken', class Errors, trigger "Main_DB_AlwaysRUN_Alarm_SurgeTankRunDry" bit 0
   18: 'Wasserstation Ausgleichsbehälter läuft über', class Errors, trigger "Main_DB_AlwaysRUN_Alarm_SurgeTankOverflow" bit 0

analog alarms
   1: 'flow temperature too high', class Warnings, trigger "Main_DB_FlowTemperaturePlant"

text list "Textliste_Bildnamen": 1 'Grundbild'; 2 'IO'; 3 'RuntimeMeters'; 4 'Settings'

Template "Vorlage_1" 1280x800
   Button "Beenden" at 1182,752 size 67x47; TextOff 'Beenden'; PictureOff "ExitRuntime_KTP1200_Basic_PN_TR"; PictureOn "ExitRuntime_KTP1200_Basic_PN_TR"
      on Release: StopRuntime(0)
   Button "Template_Button" at 1054,752 size 67x47; TextOff 'Text'
   Button "Template_Button_1" at 926,752 size 67x47; TextOff 'Text'
   Button "Template_Button_2" at 798,752 size 67x47; TextOff 'Text'
   Button "Template_Button_3" at 670,752 size 67x47; TextOff 'Text'
   Button "Template_Button_4" at 542,752 size 67x47; TextOff 'RTM'
      on Release: ActivateScreen("RuntimeMeters", 0)
   Button "Template_Button_5" at 414,752 size 67x47; TextOff 'IO'
      on Release: ActivateScreen("IO", 0)
   Button "Template_Button_6" at 286,752 size 67x47; TextOff 'OPT'
      on Release: ActivateScreen("Settings", 0)
   Button "Meldungen" at 158,752 size 67x47; TextOff 'Meldungen'; PictureOff "AlarmDisplay_KTP1200_Basic_PN_TR"; PictureOn "AlarmDisplay_KTP1200_Basic_PN_TR"
      on Release: function_ef3f5d25("Meldefenster_Nichtquittiert", -1)
   Button "Startbild" at 30,752 size 67x47; TextOff 'Startbild'; PictureOff "NavigateHome_KTP1200_Basic_PN_TR"; PictureOn "NavigateHome_KTP1200_Basic_PN_TR"
      on Release: ActivateScreen("Grundbild", 0)
   SymbolicIOField "Symbolisches_EA_Feld_Bild" at 87,9 size 1086x30; TextOff '0'; TextOn '1'; TextList "Textliste_Bildnamen"
      ProcessValue <- "Variable_Bildnummer"
      on Change: ActivateScreenByNumber("Variable_Bildnummer", 0)
   DateTimeField "HmiScreenItemData" at 1175,24 size 105x24
   DateTimeField "HmiScreenItemData_1" at 1175,0 size 105x24
   GraphicView "Logo" at 0,0 size 85x48; Picture "Logo von HMI_1"

screen "Grundbild" 1280x800, template "Vorlage_1"
   on GenerateScreen: SetTag("Variable_Bildnummer", 1)
   TextField "Textfeld_1" at 45,187 size 212x25; Text 'Vorlauftemperatur Werk / flow temperature'
   IOField "EA-Feld_1" at 326,185 size 96x32; FormatPattern s999999999.99
      ProcessValue <- "Main_DB_FlowTemperaturePlant"
   TextField "Textfeld_2" at 3,46 size 185x94; Text 'Gelsenkirchen Kühlturm +Feld1 Text Debrecen hűtőtorony +mező1'
   TextField "Textfeld_3" at 45,225 size 279x25; Text 'Vorlauftemperatur Ofenkühlung / return temperature'
   IOField "EA-Feld_2" at 326,223 size 96x32; FormatPattern s999999999.99
      ProcessValue <- "Main_DB_FlowTemperatureFurnace"
   TextField "Textfeld_4" at 424,185 size 25x25; Text '°C'
   TextField "Textfeld_5" at 424,223 size 25x25; Text '°C'
   TrendView "Kurvenanzeige_1" at 153,428 size 600x300
   Switch "Schalter_1" at 633,133 size 120x32; CaptionText 'Switch'; TextOff 'HAND'; TextOn 'AUTO'
      ProcessValue <- "Main_DB_AutoMode"
   TextField "Textfeld_6" at 821,139 size 80x25; Text 'Pumpe 1'
      Visibility <- "Main_DB_AutoMode"
   Switch "Schalter_2" at 1012,136 size 64x32; CaptionText 'Switch'; TextOff 'OFF'; TextOn 'ON'
      Visibility <- "Main_DB_AutoMode"
      ProcessValue <- "Werkspumpe 1"
   TextField "Textfeld_7" at 821,178 size 80x25; Text 'Pumpe 2'
      Visibility <- "Main_DB_AutoMode"
   Switch "Schalter_3" at 1012,176 size 64x32; TextOn 'ON'; CaptionText 'Switch'; TextOff 'OFF'
      Visibility <- "Main_DB_AutoMode"
      ProcessValue <- "Werkspumpe 2"
   Switch "Schalter_4" at 1012,216 size 64x32; TextOn 'ON'; CaptionText 'Switch'; TextOff 'OFF'
      Visibility <- "Main_DB_AutoMode"
      ProcessValue <- "Kühlwasserpumpe 1"
   Switch "Schalter_5" at 1012,256 size 64x32; TextOn 'ON'; CaptionText 'Switch'; TextOff 'OFF'
      Visibility <- "Main_DB_AutoMode"
      ProcessValue <- "Kühlwasserpumpe 2"
   Switch "Schalter_6" at 1012,296 size 64x32; TextOn 'ON'; CaptionText 'Switch'; TextOff 'OFF'
      Visibility <- "Main_DB_AutoMode"
      ProcessValue <- "KT 1 Ventilator"
   Switch "Schalter_7" at 1012,336 size 64x32; TextOn 'ON'; CaptionText 'Switch'; TextOff 'OFF'
      Visibility <- "Main_DB_AutoMode"
      ProcessValue <- "KT 2 Ventilator"
   TextField "Textfeld_8" at 821,218 size 80x25; Text 'Pumpe 3'
      Visibility <- "Main_DB_AutoMode"
   TextField "Textfeld_9" at 821,260 size 80x25; Text 'Pumpe 4'
      Visibility <- "Main_DB_AutoMode"
   TextField "Textfeld_10" at 821,299 size 105x25; Text 'Ventilator 1'
      Visibility <- "Main_DB_AutoMode"
   TextField "Textfeld_11" at 821,340 size 105x25; Text 'Ventilator 2'
      Visibility <- "Main_DB_AutoMode"
   IOField "EA-Feld_3" at 1085,295 size 50x32; FormatPattern 999
      ProcessValue <- "Main_DB_Hand_static_Vent1SollP"
      Visibility <- "Main_DB_AutoMode"
   IOField "EA-Feld_4" at 1085,335 size 50x32; FormatPattern 999
      Visibility <- "Main_DB_AutoMode"
      ProcessValue <- "Main_DB_Hand_static_Vent2SollP"
   IOField "EA-Feld_5" at 326,263 size 96x32; FormatPattern s999999999.99
      ProcessValue <- "Main_DB_Auto_s_Max"
   TextField "Textfeld_12" at 424,265 size 213x25; Text '°C default value is 27 °C'
   TextField "Textfeld_13" at 48,265 size 76x25; Text 'Sollwert / setpoint'
   TextField "Textfeld_14" at 820,378 size 186x25; Text 'Pumpe Hebeanlage 1'
      Visibility <- "Main_DB_AutoMode"
   Switch "Schalter_8" at 1011,375 size 64x32; TextOn 'ON'; CaptionText 'Switch'; TextOff 'OFF'
      Visibility <- "Main_DB_AutoMode"
      ProcessValue <- "Ofenpumpe 1"
   TextField "Textfeld_15" at 820,417 size 186x25; Text 'Pumpe Hebeanlage 2'
      Visibility <- "Main_DB_AutoMode"
   Switch "Schalter_9" at 1011,415 size 64x32; TextOn 'ON'; CaptionText 'Switch'; TextOff 'OFF'
      Visibility <- "Main_DB_AutoMode"
      ProcessValue <- "Ofenpumpe 2"
   TextField "Textfeld_16" at 820,457 size 184x25; Text 'ZU-Klappen 1 öffnen'
      Visibility <- "Main_DB_AutoMode"
   Switch "Schalter_10" at 1011,455 size 64x32; TextOn 'ON'; CaptionText 'Switch'; TextOff 'OFF'
      Visibility <- "Main_DB_AutoMode"
      ProcessValue <- "KT 1 Sprührohr-Klappen öffnen"
   TextField "Textfeld_17" at 820,497 size 184x25; Text 'ZU-Klappen 2 öffnen'
      Visibility <- "Main_DB_AutoMode"
   Switch "Schalter_11" at 1011,495 size 64x32; TextOn 'ON'; CaptionText 'Switch'; TextOff 'OFF'
      Visibility <- "Main_DB_AutoMode"
      ProcessValue <- "KT 2 Sprührohr-Klappen öffnen"
   TextField "Textfeld_18" at 820,537 size 184x25; Text 'Hebeanlage 1 öffnen'
      Visibility <- "Main_DB_AutoMode"
   Switch "Schalter_12" at 1011,535 size 64x32; TextOn 'ON'; CaptionText 'Switch'; TextOff 'OFF'
      Visibility <- "Main_DB_AutoMode"
      ProcessValue <- "HA 1 Klappe Freigabe"
   TextField "Textfeld_19" at 820,577 size 184x25; Text 'Hebeanlage 2 öffnen'
      Visibility <- "Main_DB_AutoMode"
   Switch "Schalter_13" at 1011,575 size 64x32; TextOn 'ON'; CaptionText 'Switch'; TextOff 'OFF'
      Visibility <- "Main_DB_AutoMode"
      ProcessValue <- "HA 2 Klappe Freigabe"
   TextField "Textfeld_20" at 820,617 size 148x67; Text 'Wasserbehälter Wassercontainer Nachfüllung'
      Visibility <- "Main_DB_AutoMode"
   Switch "Schalter_14" at 1011,615 size 64x32; TextOn 'ON'; CaptionText 'Switch'; TextOff 'OFF'
      Visibility <- "Main_DB_AutoMode"
      ProcessValue <- "Main_DB_HMI_StorageTankRefill"
   IOField "EA-Feld_6" at 1080,615 size 50x32; FormatPattern 999
      Visibility <- "Main_DB_AutoMode"
      ProcessValue <- "WSB OUT Byte"

screen "IO" 1280x800, template "Vorlage_1"
   TextField "Text field_1" at 20,50 size 134x20; Text 'Steuerspannung Ein'
      Appearance <- "Steuerspannung Ein"
   TextField "Text field_2" at 20,70 size 159x20; Text 'Sicherung Ausgänge OK'
      Appearance <- "Sicherung Ausgänge OK"
   TextField "Text field_3" at 20,90 size 138x20; Text 'Ventilator 1 Störung'
      Appearance <- "KT 1 Ventilator Störung"
   TextField "Text field_4" at 20,110 size 133x20; Text 'Ventilator 1 Betrieb'
      Appearance <- "KT 1 Ventilator Betrieb"
   TextField "Text field_5" at 20,130 size 229x20; Text 'Ventilator 1 Reparaturschalter ein'
      Appearance <- "KT 1 Ventilator RS"
   TextField "Text field_6" at 20,150 size 138x20; Text 'Ventilator 2 Störung'
      Appearance <- "KT 2 Ventilator Störung"
   TextField "Text field_7" at 20,170 size 133x20; Text 'Ventilator 2 Betrieb'
      Appearance <- "KT 2 Ventilator Betrieb"
   TextField "Text field_8" at 20,190 size 229x20; Text 'Ventilator 2 Reparaturschalter ein'
      Appearance <- "KT 2 Ventilator RS"
   TextField "Text field_9" at 20,210 size 116x20; Text 'Störung Pumpe 1'
      Appearance <- "Werkspumpe 1 Störung"
   TextField "Text field_10" at 20,230 size 111x20; Text 'Betrieb Pumpe 1'
      Appearance <- "Werkspumpe 1 Betrieb"
   TextField "Text field_11" at 20,250 size 116x20; Text 'Störung Pumpe 2'
      Appearance <- "Werkspumpe 2 Störung"
   TextField "Text field_12" at 20,270 size 111x20; Text 'Betrieb Pumpe 2'
      Appearance <- "Werkspumpe 2 Betrieb"
   TextField "Text field_13" at 20,290 size 41x20; Text 'XXXX'
      Appearance <- "Reserve DI1.4"
   TextField "Text field_14" at 20,310 size 81x20; Text 'RESERVE(1)'
      Appearance <- "Reserve DI1.5"
   TextField "Text field_15" at 20,330 size 82x20; Text 'Ventilator 1'
      Appearance <- "KT 1 Ventilator"
   TextField "Text field_16" at 20,350 size 82x20; Text 'Ventilator 2'
      Appearance <- "KT 2 Ventilator"
   TextField "Text field_17" at 20,370 size 60x20; Text 'Pumpe 1'
      Appearance <- "Werkspumpe 1"
   TextField "Text field_18" at 20,390 size 60x20; Text 'Pumpe 2'
      Appearance <- "Werkspumpe 2"
   TextField "Text field_19" at 20,410 size 60x20; Text 'Pumpe 3'
      Appearance <- "Kühlwasserpumpe 1"
   TextField "Text field_20" at 20,430 size 60x20; Text 'Pumpe 4'
      Appearance <- "Kühlwasserpumpe 2"
   TextField "Text field_22" at 20,450 size 161x20; Text 'Rundumleuchte Störung'
      Appearance <- "Rundumleuchte Störung"
   TextField "Text field_23" at 20,470 size 93x20; Text 'Reserve DQ 1'
      Appearance <- "Reserve DQ0.7"
   TextField "Text field_24" at 20,490 size 135x20; Text 'ZU-Klappen 1 öffnen'
      Appearance <- "KT 1 Sprührohr-Klappen öffnen"
   TextField "Text field_25" at 20,510 size 135x20; Text 'ZU-Klappen 2 öffnen'
      Appearance <- "KT 2 Sprührohr-Klappen öffnen"
   TextField "Text field_26" at 270,50 size 220x20; Text 'Motorschutzschalter Pumpe 3 OK'
      Appearance <- "Kühlwasserpumpe 1 MSS OK"
   TextField "Text field_27" at 270,70 size 220x20; Text 'Motorschutzschalter Pumpe 4 OK'
      Appearance <- "Kühlwasserpumpe 2 MSS OK"
   TextField "Text field_28" at 270,90 size 232x20; Text 'Motorschutzschalter Hebeanlage 1'
      Appearance <- "Ofenpumpe 1 MSS OK"
   TextField "Text field_29" at 270,110 size 232x20; Text 'Motorschutzschalter Hebeanlage 2'
      Appearance <- "Ofenpumpe 2 MSS OK"
   TextField "Text field_30" at 270,130 size 111x20; Text 'Betrieb Pumpe 3'
      Appearance <- "Kühlwasserpumpe 1 Betrieb"
   TextField "Text field_31" at 270,150 size 111x20; Text 'Betrieb Pumpe 4'
      Appearance <- "Kühlwasserpumpe 2 Betrieb"
   TextField "Text field_32" at 270,170 size 191x20; Text 'Betrieb Pumpe Hebeanlage 1'
      Appearance <- "Ofenpumpe 1 Betrieb"
   TextField "Text field_33" at 270,190 size 191x20; Text 'Betrieb Pumpe Hebeanlage 2'
      Appearance <- "Ofenpumpe 2 Betrieb"
   TextField "Text field_34" at 270,210 size 149x20; Text 'ZU-Klappen 1 geöffnet'
      Appearance <- "KT 1 Sprührohr-Klappen geöffnet"
   TextField "Text field_35" at 270,230 size 149x20; Text 'ZU-Klappen 2 geöffnet'
      Appearance <- "KT 2 Sprührohr-Klappen geöffnet"
   TextField "Text field_36" at 270,250 size 200x20; Text 'Hebeanlage 1 Klappe geöffnet'
      Appearance <- "HA 1 Klappe geöffnet"
   TextField "Text field_37" at 270,270 size 223x20; Text 'Hebeanlage 1 Klappe geschlossen'
      Appearance <- "HA 1 Klappe geschlossen"
   TextField "Text field_38" at 270,290 size 200x20; Text 'Hebeanlage 2 Klappe geöffnet'
      Appearance <- "HA 2 Klappe geöffnet"
   TextField "Text field_39" at 270,310 size 223x20; Text 'Hebeanlage 2 Klappe geschlossen'
      Appearance <- "HA 2 Klappe geschlossen"
   TextField "Text field_40" at 270,330 size 97x20; Text 'Reserve DI 22'
      Appearance <- "Reserve DI9.6"
   TextField "Text field_41" at 270,350 size 97x20; Text 'Reserve DI 23'
      Appearance <- "Reserve DI9.7"
   TextField "Text field_42" at 270,370 size 139x20; Text 'Hebeanlage 1 öffnen'
      Appearance <- "HA 1 Klappe Freigabe"
   TextField "Text field_43" at 270,390 size 139x20; Text 'Hebeanlage 2 öffnen'
      Appearance <- "HA 2 Klappe Freigabe"
   TextField "Text field_44" at 270,410 size 140x20; Text 'Pumpe Hebeanlage 1'
      Appearance <- "Ofenpumpe 1"
   TextField "Text field_45" at 270,430 size 140x20; Text 'Pumpe Hebeanlage 2'
      Appearance <- "Ofenpumpe 2"
   TextField "Text field_46" at 270,450 size 93x20; Text 'Reserve DQ 2'
      Appearance <- "Reserve DQ8.4"
   TextField "Text field_47" at 270,470 size 93x20; Text 'Reserve DQ 3'
      Appearance <- "Reserve DQ8.5"
   TextField "Text field_48" at 270,490 size 93x20; Text 'Reserve DQ 4'
      Appearance <- "Reserve DQ8.6"
   TextField "Text field_49" at 270,510 size 93x20; Text 'Reserve DQ 5'
      Appearance <- "Reserve DQ8.7"
   TextField "Text field_50" at 270,530 size 302x20; Text 'Wasserbehälter Wassercontainer Nachfüllung'
      Appearance <- "WSB Magnetventil"
   TextField "Text field_51" at 270,550 size 93x20; Text 'Reserve DQ 7'
      Appearance <- "Reserve DQ9.1"
   TextField "Text field_52" at 270,570 size 93x20; Text 'Reserve DQ 8'
      Appearance <- "Reserve DQ9.2"
   TextField "Text field_53" at 270,590 size 93x20; Text 'Reserve DQ 9'
      Appearance <- "Reserve DQ9.3"
   TextField "Text field_54" at 270,610 size 101x20; Text 'Reserve DQ 10'
      Appearance <- "Reserve DQ9.4"
   TextField "Text field_55" at 270,630 size 101x20; Text 'Reserve DQ 11'
      Appearance <- "Reserve DQ9.5"
   TextField "Text field_56" at 270,650 size 101x20; Text 'Reserve DQ 12'
      Appearance <- "Reserve DQ9.6"
   TextField "Text field_57" at 270,670 size 101x20; Text 'Reserve DQ 13'
      Appearance <- "Reserve DQ9.7"
   TextField "Text field_58" at 550,50 size 137x20; Text 'Absalzanlage Impuls'
      Appearance <- "Absalzanlage läuft"
   TextField "Text field_59" at 550,70 size 145x20; Text 'Wasserbehälter OUT1'
      Appearance <- "WSB OUT1"
   TextField "Text field_60" at 550,90 size 145x20; Text 'Wasserbehälter OUT2'
      Appearance <- "WSB OUT2"
   TextField "Text field_61" at 550,110 size 145x20; Text 'Wasserbehälter OUT3'
      Appearance <- "WSB OUT3"
   TextField "Text field_62" at 550,130 size 145x20; Text 'Wasserbehälter OUT4'
      Appearance <- "WSB OUT4"
   TextField "Text field_63" at 550,150 size 89x20; Text 'Reserve DI 9'
      Appearance <- "Reserve DI12.5"
   TextField "Text field_64" at 550,170 size 97x20; Text 'Reserve DI 10'
      Appearance <- "Reserve DI12.6"
   TextField "Text field_65" at 550,190 size 97x20; Text 'Reserve DI 11'
      Appearance <- "Reserve DI12.7"
   TextField "Text field_66" at 550,210 size 97x20; Text 'Reserve DI 12'
      Appearance <- "Reserve DI13.0"
   TextField "Text field_67" at 550,230 size 97x20; Text 'Reserve DI 13'
      Appearance <- "Reserve DI13.1"
   TextField "Text field_68" at 550,250 size 97x20; Text 'Reserve DI 14'
      Appearance <- "Reserve DI13.2"
   TextField "Text field_69" at 550,270 size 97x20; Text 'Reserve DI 15'
      Appearance <- "Reserve DI13.3"
   TextField "Text field_70" at 550,290 size 97x20; Text 'Reserve DI 16'
      Appearance <- "Reserve DI13.4"
   TextField "Text field_71" at 550,310 size 97x20; Text 'Reserve DI 17'
      Appearance <- "Reserve DI13.5"
   TextField "Text field_72" at 550,330 size 97x20; Text 'Reserve DI 18'
      Appearance <- "Reserve DI13.6"
   TextField "Text field_73" at 550,350 size 97x20; Text 'Reserve DI 19'
      Appearance <- "Reserve DI13.7"
   TextField "Text field_74" at 720,50 size 127x20; Text 'Vorlauftemperatur'
   TextField "Text field_75" at 720,90 size 143x20; Text 'Ruecklauftemperatur'
   TextField "Text field_76" at 720,130 size 192x20; Text 'Hebeanlage 1 Differenzdruck'
   TextField "Text field_77" at 720,170 size 192x20; Text 'Hebeanlage 2 Differenzdruck'
   TextField "Text field_78" at 720,210 size 93x20; Text 'Reserve IW 1'
   TextField "Text field_79" at 720,250 size 93x20; Text 'Reserve IW 2'
   TextField "Text field_80" at 720,290 size 139x20; Text 'Sollwert Ventilator 1'
   TextField "Text field_81" at 720,330 size 139x20; Text 'Sollwert Ventilator 2'
   TextField "Text field_82" at 720,370 size 202x20; Text 'Hebeanlage 1 Durchflußmenge'
   TextField "Text field_83" at 720,410 size 202x20; Text 'Hebeanlage 2 Durchflußmenge'
   IOField "I/O field_1" at 950,50 size 63x20; FormatPattern s999999
      ProcessValue <- "Vorlauftemperatur Werk"
   IOField "I/O field_2" at 950,90 size 63x20; FormatPattern s999999
      ProcessValue <- "Vorlauftemperatur Ofen"
   IOField "I/O field_3" at 950,130 size 63x20; FormatPattern s999999
      ProcessValue <- "HA 1 Differenzdruck"
   IOField "I/O field_4" at 950,170 size 63x20; FormatPattern s999999
      ProcessValue <- "HA 2 Differenzdruck"
   IOField "I/O field_5" at 950,210 size 55x20; FormatPattern s99999
      ProcessValue <- "Reserve IW132"
   IOField "I/O field_6" at 950,250 size 63x20; FormatPattern s999999
      ProcessValue <- "Reserve IW134"
   IOField "I/O field_7" at 950,290 size 63x20; FormatPattern s999999
      ProcessValue <- "KT 1 Ventilator Sollwert"
   IOField "I/O field_8" at 950,330 size 63x20; FormatPattern s999999
      ProcessValue <- "KT 2 Ventilator Sollwert"
   IOField "I/O field_9" at 950,370 size 63x20; FormatPattern s999999
      ProcessValue <- "HA 1 Klappe Durchflußmenge"
   IOField "I/O field_10" at 950,410 size 63x20; FormatPattern s999999
      ProcessValue <- "HA 2 Klappe Durchflußmenge"
   IOField "I/O field_11" at 1020,50 size 47x20; FormatPattern s9999
      ProcessValue <- "Vorlauftemperatur Werk(1)"
   IOField "I/O field_12" at 1020,90 size 47x20; FormatPattern s9999
      ProcessValue <- "Vorlauftemperatur Ofen(1)"
   IOField "I/O field_13" at 1020,130 size 47x20; FormatPattern s9999
      ProcessValue <- "HA 1 Differenzdruck(1)"
   IOField "I/O field_14" at 1020,170 size 47x20; FormatPattern s9999
      ProcessValue <- "HA 2 Differenzdruck(1)"
   IOField "I/O field_15" at 1020,210 size 47x20; FormatPattern s9999
      ProcessValue <- "Reserve IW132(1)"
   IOField "I/O field_16" at 1020,250 size 47x20; FormatPattern s9999
      ProcessValue <- "Reserve IW134(1)"
   IOField "I/O field_17" at 1020,290 size 47x20; FormatPattern s9999
      ProcessValue <- "KT 1 Ventilator Sollwert(1)"
   IOField "I/O field_18" at 1020,330 size 47x20; FormatPattern s9999
      ProcessValue <- "KT 2 Ventilator Sollwert(1)"
   IOField "I/O field_19" at 1020,370 size 47x20; FormatPattern s9999
      ProcessValue <- "HA 1 Klappe Durchflußmenge(1)"
   IOField "I/O field_20" at 1020,410 size 47x20; FormatPattern s9999
      ProcessValue <- "HA 2 Klappe Durchflußmenge(1)"
   Bar "Bar_1" at 1075,50 size 200x40; MinimumValue 0; MaximumValue 100
      ProcessValue <- "Vorlauftemperatur Werk(1)"
   Bar "Bar_2" at 1075,90 size 200x40; MinimumValue 0; MaximumValue 100
      ProcessValue <- "Vorlauftemperatur Ofen(1)"
   Bar "Bar_3" at 1075,130 size 200x40; MinimumValue 0; MaximumValue 100
      ProcessValue <- "HA 1 Differenzdruck(1)"
   Bar "Bar_4" at 1075,170 size 200x40; MinimumValue 0; MaximumValue 100
      ProcessValue <- "HA 2 Differenzdruck(1)"
   Bar "Bar_5" at 1075,210 size 200x40; MinimumValue 0; MaximumValue 100
      ProcessValue <- "Reserve IW132(1)"
   Bar "Bar_6" at 1075,250 size 200x40; MinimumValue 0; MaximumValue 100
      ProcessValue <- "Reserve IW134(1)"
   Bar "Bar_7" at 1075,290 size 200x40; MinimumValue 0; MaximumValue 100
      ProcessValue <- "KT 1 Ventilator Sollwert(1)"
   Bar "Bar_8" at 1075,330 size 200x40; MinimumValue 0; MaximumValue 100
      ProcessValue <- "KT 2 Ventilator Sollwert(1)"
   Bar "Bar_9" at 1075,370 size 200x40; MinimumValue 0; MaximumValue 100
      ProcessValue <- "HA 1 Klappe Durchflußmenge(1)"
   Bar "Bar_10" at 1075,410 size 200x40; MinimumValue 0; MaximumValue 100
      ProcessValue <- "HA 2 Klappe Durchflußmenge(1)"

screen "RuntimeMeters" 1280x800, template "Vorlage_1"
   TextField "Text field_1" at 50,100 size 38x25; Text 'SPS / PLC'
   TextField "Text field_2" at 50,125 size 147x25; Text 'Betrieb Pumpe 1'
   TextField "Text field_3" at 50,150 size 147x25; Text 'Betrieb Pumpe 2'
   TextField "Text field_4" at 50,175 size 147x25; Text 'Betrieb Pumpe 3'
   TextField "Text field_5" at 50,200 size 147x25; Text 'Betrieb Pumpe 4'
   TextField "Text field_6" at 50,225 size 186x25; Text 'Pumpe Hebeanlage 1'
   TextField "Text field_7" at 50,250 size 186x25; Text 'Pumpe Hebeanlage 2'
   TextField "Text field_8" at 50,275 size 172x25; Text 'Ventilator 1 Betrieb'
   TextField "Text field_9" at 50,300 size 172x25; Text 'Ventilator 2 Betrieb'
   TextField "Text field_10" at 50,325 size 53x25; Text 'RTM9'
   IOField "I/O field_1" at 300,100 size 128x25; FormatPattern s9999999999
      ProcessValue <- "Main_DB_AlwaysRUN_RuntimeMeters_SRTM{0}_s_CV"
   IOField "I/O field_2" at 300,125 size 128x25; FormatPattern s9999999999
      ProcessValue <- "Main_DB_AlwaysRUN_RuntimeMeters_SRTM{1}_s_CV"
   IOField "I/O field_3" at 300,150 size 128x25; FormatPattern s9999999999
      ProcessValue <- "Main_DB_AlwaysRUN_RuntimeMeters_SRTM{2}_s_CV"
   IOField "I/O field_4" at 300,175 size 128x25; FormatPattern s9999999999
      ProcessValue <- "Main_DB_AlwaysRUN_RuntimeMeters_SRTM{3}_s_CV"
   IOField "I/O field_5" at 300,200 size 128x25; FormatPattern s9999999999
      ProcessValue <- "Main_DB_AlwaysRUN_RuntimeMeters_SRTM{4}_s_CV"
   IOField "I/O field_6" at 300,225 size 128x25; FormatPattern s9999999999
      ProcessValue <- "Main_DB_AlwaysRUN_RuntimeMeters_SRTM{5}_s_CV"
   IOField "I/O field_7" at 300,250 size 128x25; FormatPattern s9999999999
      ProcessValue <- "Main_DB_AlwaysRUN_RuntimeMeters_SRTM{6}_s_CV"
   IOField "I/O field_8" at 300,275 size 128x25; FormatPattern s9999999999
      ProcessValue <- "Main_DB_AlwaysRUN_RuntimeMeters_SRTM{7}_s_CV"
   IOField "I/O field_9" at 300,300 size 128x25; FormatPattern s9999999999
      ProcessValue <- "Main_DB_AlwaysRUN_RuntimeMeters_SRTM{8}_s_CV"
   IOField "I/O field_10" at 300,325 size 128x25; FormatPattern s9999999999
      ProcessValue <- "Main_DB_AlwaysRUN_RuntimeMeters_SRTM{9}_s_CV"
   IOField "I/O field_11" at 440,100 size 18x25; FormatPattern 1
      ProcessValue <- "Main_DB_AlwaysRUN_RuntimeMeters_SRTM{0}_s_CQ"
   IOField "I/O field_12" at 440,125 size 18x25; FormatPattern 1
      ProcessValue <- "Main_DB_AlwaysRUN_RuntimeMeters_SRTM{1}_s_CQ"
   IOField "I/O field_13" at 440,150 size 18x25; FormatPattern 1
      ProcessValue <- "Main_DB_AlwaysRUN_RuntimeMeters_SRTM{2}_s_CQ"
   IOField "I/O field_14" at 440,175 size 18x25; FormatPattern 1
      ProcessValue <- "Main_DB_AlwaysRUN_RuntimeMeters_SRTM{3}_s_CQ"
   IOField "I/O field_15" at 440,200 size 18x25; FormatPattern 1
      ProcessValue <- "Main_DB_AlwaysRUN_RuntimeMeters_SRTM{4}_s_CQ"
   IOField "I/O field_16" at 440,225 size 18x25; FormatPattern 1
      ProcessValue <- "Main_DB_AlwaysRUN_RuntimeMeters_SRTM{5}_s_CQ"
   IOField "I/O field_17" at 440,250 size 18x25; FormatPattern 1
      ProcessValue <- "Main_DB_AlwaysRUN_RuntimeMeters_SRTM{6}_s_CQ"
   IOField "I/O field_18" at 440,275 size 18x25; FormatPattern 1
      ProcessValue <- "Main_DB_AlwaysRUN_RuntimeMeters_SRTM{7}_s_CQ"
   IOField "I/O field_19" at 440,300 size 18x25; FormatPattern 1
      ProcessValue <- "Main_DB_AlwaysRUN_RuntimeMeters_SRTM{8}_s_CQ"
   IOField "I/O field_20" at 440,325 size 18x25; FormatPattern 1
      ProcessValue <- "Main_DB_AlwaysRUN_RuntimeMeters_SRTM{9}_s_CQ"
   IOField "I/O field_21" at 490,100 size 18x25; FormatPattern 1
      ProcessValue <- "Main_DB_AlwaysRUN_RuntimeMeters_SRTM{0}_i_CLK"
   IOField "I/O field_22" at 490,125 size 18x25; FormatPattern 1
      ProcessValue <- "Main_DB_AlwaysRUN_RuntimeMeters_SRTM{1}_i_CLK"
   IOField "I/O field_23" at 490,150 size 18x25; FormatPattern 1
      ProcessValue <- "Main_DB_AlwaysRUN_RuntimeMeters_SRTM{2}_i_CLK"
   IOField "I/O field_24" at 490,175 size 18x25; FormatPattern 1
      ProcessValue <- "Main_DB_AlwaysRUN_RuntimeMeters_SRTM{3}_i_CLK"
   IOField "I/O field_25" at 490,200 size 18x25; FormatPattern 1
      ProcessValue <- "Main_DB_AlwaysRUN_RuntimeMeters_SRTM{4}_i_CLK"
   IOField "I/O field_26" at 490,225 size 18x25; FormatPattern 1
      ProcessValue <- "Main_DB_AlwaysRUN_RuntimeMeters_SRTM{5}_i_CLK"
   IOField "I/O field_27" at 490,250 size 18x25; FormatPattern 1
      ProcessValue <- "Main_DB_AlwaysRUN_RuntimeMeters_SRTM{6}_i_CLK"
   IOField "I/O field_28" at 490,275 size 18x25; FormatPattern 1
      ProcessValue <- "Main_DB_AlwaysRUN_RuntimeMeters_SRTM{7}_i_CLK"
   IOField "I/O field_29" at 490,300 size 18x25; FormatPattern 1
      ProcessValue <- "Main_DB_AlwaysRUN_RuntimeMeters_SRTM{8}_i_CLK"
   IOField "I/O field_30" at 490,325 size 18x25; FormatPattern 1
      ProcessValue <- "Main_DB_AlwaysRUN_RuntimeMeters_SRTM{9}_i_CLK"
   TextField "Text field_11" at 300,75 size 27x25; Text 'CV'
   TextField "Text field_12" at 440,75 size 29x25; Text 'CQ'
   TextField "Text field_13" at 490,75 size 38x25; Text 'CLK'

screen "Settings" 1280x800, template "Vorlage_1"
   TextField "Textfeld_20" at 40,65 size 148x67; Text 'Wasserbehälter Wassercontainer Nachfüllung'
      Visibility <- "Main_DB_AutoMode"
   TextField "Textfeld_1" at 45,165 size 42x25; Text 'P1'
      Visibility <- "Main_DB_AutoMode"
   TextField "Textfeld_2" at 45,195 size 42x25; Text 'P2'
      Visibility <- "Main_DB_AutoMode"
   TextField "Textfeld_3" at 45,230 size 42x25; Text 'P3'
      Visibility <- "Main_DB_AutoMode"
   TextField "Textfeld_4" at 45,265 size 42x25; Text 'P4'
      Visibility <- "Main_DB_AutoMode"
   IOField "I/O field_1" at 100,165 size 96x32; FormatPattern s99999
      ProcessValue <- "Main_DB_HMI_StorageTankLevel_P1"
   IOField "I/O field_2" at 100,200 size 96x32; FormatPattern s99999
      ProcessValue <- "Main_DB_HMI_StorageTankLevel_P2"
   IOField "I/O field_3" at 100,235 size 96x32; FormatPattern s99999
      ProcessValue <- "Main_DB_HMI_StorageTankLevel_P3"
   IOField "I/O field_4" at 100,270 size 96x32; FormatPattern s99999
      ProcessValue <- "Main_DB_HMI_StorageTankLevel_P4"
*)